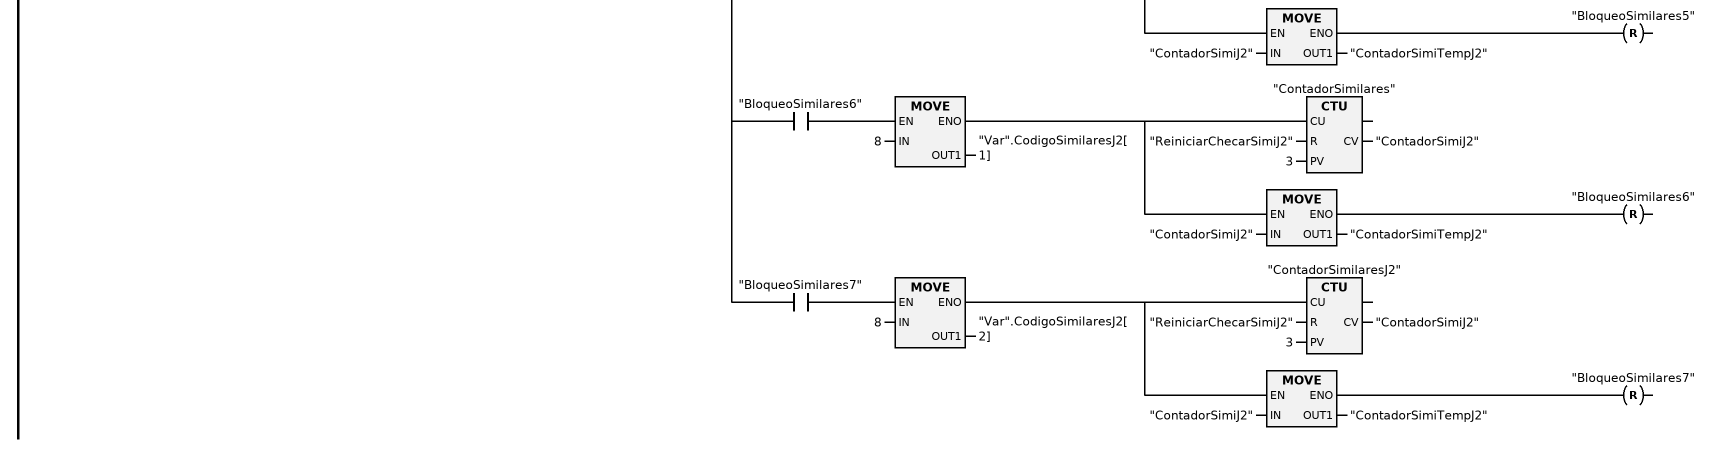
   #_w1 := "Panel1AzulJ2" AND ("Var".VectorPrincipalJ2["IntentoCompletoJ2", 0] = 0) AND "Bounce6";
   IF #_w1 THEN
       "Var".VectorPrincipalJ2["IntentoCompletoJ2", 0] := 5;
       "Intento0J2" := TRUE;
   END_IF;
   #_w2 := #_w1 AND ("Var".VectorPrincipalJ2["IntentoCompletoJ2", 0] = "Var".CodigoOJ2[0]);
   "ContadorCorrectasJ2".CTU(CU := #_w2, R := "ReiniciarChecarCorrJ2", PV := 3, CV => "ContadorCorrJ2");
   IF #_w2 THEN
       "ContadorCorrTempJ2" := "ContadorCorrJ2";
       "Var".CodigoSimilaresJ2[0] := 8;
       "BloqueoSimilares8" := TRUE;
   END_IF;
   #_w3 := #_w2 AND ("Var".CodigoSimilaresJ2[0] = 8);
   "ContadorSimilaresJ2".CTD(CD := #_w3, LD := "ReiniciarChecarSimiJ2", PV := 3, CV => "ContadorSimiJ2");
   IF #_w3 THEN "ContadorSimiTempJ2" := "ContadorSimiJ2"; END_IF;
   #_w4 := #_w1 AND NOT "BloqueoSimilares8" AND ("Var".VectorPrincipalJ2["IntentoCompletoJ2", 0] <> "Var".CodigoOJ2[0]);
   IF #_w4 AND ("Var".VectorPrincipalJ2["IntentoCompletoJ2", 0] = "Var".CodigoSimilaresJ2[1]) THEN
       "BloqueoSimilares5" := TRUE;
   END_IF;
   #_w5 := #_w4 AND ("Var".VectorPrincipalJ2["IntentoCompletoJ2", 0] <> "Var".CodigoSimilaresJ2[1]);
   IF #_w5 AND ("Var".VectorPrincipalJ2["IntentoCompletoJ2", 0] = "Var".CodigoSimilaresJ2[2]) THEN
       "BloqueoSimilares6" := TRUE;
   END_IF;
   IF #_w5 AND ("Var".VectorPrincipalJ2["IntentoCompletoJ2", 0] <> "Var".CodigoSimilaresJ2[2]) AND ("Var".VectorPrincipalJ2["IntentoCompletoJ2", 0] = "Var".CodigoSimilaresJ2[3]) THEN
       "BloqueoSimilares7" := TRUE;
   END_IF;
   #_w6 := #_w1 AND "BloqueoSimilares5";
   IF #_w6 THEN "Var".CodigoSimilaresJ2[1] := 8; END_IF;
   "ContadorSimilaresJ2".CTU(CU := #_w6, R := "ReiniciarChecarSimiJ2", PV := 3, CV => "ContadorSimiJ2");
   IF #_w6 THEN
       "ContadorSimiTempJ2" := "ContadorSimiJ2";
       "BloqueoSimilares5" := FALSE;
   END_IF;
   #_w7 := #_w1 AND "BloqueoSimilares6";
   IF #_w7 THEN "Var".CodigoSimilaresJ2[2] := 8; END_IF;
   "ContadorSimilaresJ2".CTU(CU := #_w7, R := "ReiniciarChecarSimiJ2", PV := 3, CV => "ContadorSimiJ2");
   IF #_w7 THEN
       "ContadorSimiTempJ2" := "ContadorSimiJ2";
       "BloqueoSimilares6" := FALSE;
   END_IF;
   #_w8 := #_w1 AND "BloqueoSimilares7";
   IF #_w8 THEN "Var".CodigoSimilaresJ2[3] := 8; END_IF;
   "ContadorSimilaresJ2".CTU(CU := #_w8, R := "ReiniciarChecarSimiJ2", PV := 3, CV => "ContadorSimiJ2");
   IF #_w8 THEN
       "ContadorSimiTempJ2" := "ContadorSimiJ2";
       "BloqueoSimilares7" := FALSE;
   END_IF;
   #_w9 := "Panel1AzulJ2" AND "Bounce7" AND "Panel1AzulJ2" AND "Intento0J2" AND ("Var".VectorPrincipalJ2["IntentoCompletoJ2", 1] = 0);
   IF #_w9 THEN
       "Var".VectorPrincipalJ2["IntentoCompletoJ2", 1] := 5;
       "Intento1J2" := TRUE;
   END_IF;
   #_w10 := #_w9 AND ("Var".VectorPrincipalJ2["IntentoCompletoJ2", 1] = "Var".CodigoOJ2[1]);
   "ContadorCorrectasJ2".CTU(CU := #_w10, R := "ReiniciarChecarCorrJ2", PV := 3, CV => "ContadorCorrJ2");
   IF #_w10 THEN
       "ContadorCorrTempJ2" := "ContadorCorrJ2";
       "Var".CodigoSimilaresJ2[1] := 8;
       "BloqueoSimilares8" := TRUE;
   END_IF;
   #_w11 := #_w10 AND ("Var".CodigoSimilaresJ2[1] = 8);
   "ContadorSimilaresJ2".CTD(CD := #_w11, LD := "ReiniciarChecarSimiJ2", PV := 3, CV => "ContadorSimiJ2");
   IF #_w11 THEN "ContadorSimiTempJ2" := "ContadorSimiJ2"; END_IF;
   #_w12 := #_w9 AND NOT "BloqueoSimilares8" AND ("Var".VectorPrincipalJ2["IntentoCompletoJ2", 1] <> "Var".CodigoOJ2[1]);
   IF #_w12 AND ("Var".VectorPrincipalJ2["IntentoCompletoJ2", 1] = "Var".CodigoSimilaresJ2[0]) THEN
       "BloqueoSimilares5" := TRUE;
   END_IF;
   #_w13 := #_w12 AND ("Var".VectorPrincipalJ2["IntentoCompletoJ2", 1] <> "Var".CodigoSimilaresJ2[0]);
   IF #_w13 AND ("Var".VectorPrincipalJ2["IntentoCompletoJ2", 1] = "Var".CodigoSimilaresJ2[2]) THEN
       "BloqueoSimilares6" := TRUE;
   END_IF;
   IF #_w13 AND ("Var".VectorPrincipalJ2["IntentoCompletoJ2", 1] <> "Var".CodigoSimilaresJ2[2]) AND ("Var".VectorPrincipalJ2["IntentoCompletoJ2", 1] = "Var".CodigoSimilaresJ2[3]) THEN
       "BloqueoSimilares7" := TRUE;
   END_IF;
   #_w14 := #_w9 AND "BloqueoSimilares5";
   IF #_w14 THEN "Var".CodigoSimilaresJ2[0] := 8; END_IF;
   "ContadorSimilaresJ2".CTU(CU := #_w14, R := "ReiniciarChecarSimiJ2", PV := 3, CV => "ContadorSimiJ2");
   IF #_w14 THEN
       "ContadorSimiTempJ2" := "ContadorSimiJ2";
       "BloqueoSimilares5" := FALSE;
   END_IF;
   #_w15 := #_w9 AND "BloqueoSimilares6";
   IF #_w15 THEN "Var".CodigoSimilaresJ1[2] := 8; END_IF;
   "ContadorSimilaresJ2".CTU(CU := #_w15, R := "ReiniciarChecarSimiJ2", PV := 3, CV => "ContadorSimiJ2");
   IF #_w15 THEN
       "ContadorSimiTempJ2" := "ContadorSimiJ2";
       "BloqueoSimilares6" := FALSE;
   END_IF;
   #_w16 := #_w9 AND "BloqueoSimilares7";
   IF #_w16 THEN "Var".CodigoSimilaresJ2[3] := 8; END_IF;
   "ContadorSimilaresJ2".CTU(CU := #_w16, R := "ReiniciarChecarSimiJ2", PV := 3, CV => "ContadorSimiJ2");
   IF #_w16 THEN
       "ContadorSimiTempJ2" := "ContadorSimiJ2";
       "BloqueoSimilares3" := FALSE;
   END_IF;
   #_w17 := "Panel1AzulJ2" AND "Bounce8" AND "Panel1AzulJ2" AND "Intento1J2" AND ("Var".VectorPrincipalJ2["IntentoCompletoJ2", 2] = 0);
   IF #_w17 THEN
       "Var".VectorPrincipalJ2["IntentoCompletoJ2", 2] := 5;
       "Intento2J2" := TRUE;
   END_IF;
   #_w18 := #_w17 AND ("Var".VectorPrincipalJ2["IntentoCompletoJ2", 2] = "Var".CodigoOJ2[2]);
   "ContadorCorrectasJ2".CTU(CU := #_w18, R := "ReiniciarChecarCorrJ2", PV := 3, CV => "ContadorCorrJ2");
   IF #_w18 THEN
       "ContadorCorrTempJ2" := "ContadorCorrJ2";
       "Var".CodigoSimilaresJ2[2] := 8;
       "BloqueoSimilares8" := TRUE;
   END_IF;
   #_w19 := #_w18 AND ("Var".CodigoSimilaresJ2[2] = 8);
   "ContadorSimilaresJ2".CTD(CD := #_w19, LD := "ReiniciarChecarSimiJ2", PV := 3, CV => "ContadorSimiJ2");
   IF #_w19 THEN "ContadorSimiTempJ2" := "ContadorSimiJ2"; END_IF;
   #_w20 := #_w17 AND NOT "BloqueoSimilares8" AND ("Var".VectorPrincipalJ2["IntentoCompletoJ2", 2] <> "Var".CodigoOJ2[2]);
   IF #_w20 AND ("Var".VectorPrincipalJ2["IntentoCompletoJ2", 2] = "Var".CodigoSimilaresJ2[0]) THEN
       "BloqueoSimilares5" := TRUE;
   END_IF;
   #_w21 := #_w20 AND ("Var".VectorPrincipalJ2["IntentoCompletoJ2", 2] <> "Var".CodigoSimilaresJ2[0]);
   IF #_w21 AND ("Var".VectorPrincipalJ2["IntentoCompletoJ2", 2] = "Var".CodigoSimilaresJ2[1]) THEN
       "BloqueoSimilares6" := TRUE;
   END_IF;
   IF #_w21 AND ("Var".VectorPrincipalJ2["IntentoCompletoJ2", 2] <> "Var".CodigoSimilaresJ2[1]) AND ("Var".VectorPrincipalJ2["IntentoCompletoJ2", 2] = "Var".CodigoSimilaresJ2[3]) THEN
       "BloqueoSimilares7" := TRUE;
   END_IF;
   #_w22 := #_w17 AND "BloqueoSimilares5";
   IF #_w22 THEN "Var".CodigoSimilaresJ2[0] := 8; END_IF;
   "ContadorSimilaresJ2".CTU(CU := #_w22, R := "ReiniciarChecarSimiJ2", PV := 3, CV => "ContadorSimiJ2");
   IF #_w22 THEN
       "ContadorSimiTempJ2" := "ContadorSimiJ2";
       "BloqueoSimilares5" := FALSE;
   END_IF;
   #_w23 := #_w17 AND "BloqueoSimilares6";
   IF #_w23 THEN "Var".CodigoSimilaresJ2[1] := 8; END_IF;
   "ContadorSimilaresJ2".CTU(CU := #_w23, R := "ReiniciarChecarSimiJ2", PV := 3, CV => "ContadorSimiJ2");
   IF #_w23 THEN
       "ContadorSimiTempJ2" := "ContadorSimiJ2";
       "BloqueoSimilares6" := FALSE;
   END_IF;
   #_w24 := #_w17 AND "BloqueoSimilares7";
   IF #_w24 THEN "Var".CodigoSimilaresJ2[3] := 8; END_IF;
   "ContadorSimilaresJ2".CTU(CU := #_w24, R := "ReiniciarChecarSimiJ2", PV := 3, CV => "ContadorSimiJ2");
   IF #_w24 THEN
       "ContadorSimiTempJ2" := "ContadorSimiJ2";
       "BloqueoSimilares7" := FALSE;
   END_IF;
   #_w25 := "Panel1AzulJ2" AND "Bounce9" AND "Panel1AzulJ2" AND "Intento2J2" AND ("Var".VectorPrincipalJ2["IntentoCompletoJ2", 3] = 0);
   IF #_w25 THEN
       "Var".VectorPrincipalJ2["IntentoCompletoJ2", 3] := 5;
       "Intento3J2" := TRUE;
   END_IF;
   #_w26 := #_w25 AND ("Var".VectorPrincipalJ2["IntentoCompletoJ2", 3] = "Var".CodigoOJ2[3]);
   "ContadorCorrectasJ2".CTU(CU := #_w26, R := "ReiniciarChecarCorrJ2", PV := 3, CV => "ContadorCorrJ2");
   IF #_w26 THEN
       "ContadorCorrTempJ2" := "ContadorCorrJ2";
       "Var".CodigoSimilaresJ2[3] := 8;
       "BloqueoSimilares8" := TRUE;
   END_IF;
   #_w27 := #_w26 AND ("Var".CodigoSimilaresJ2[3] = 8);
   "ContadorSimilaresJ2".CTD(CD := #_w27, LD := "ReiniciarChecarSimiJ2", PV := 3, CV => "ContadorSimiJ2");
   IF #_w27 THEN "ContadorSimiTempJ2" := "ContadorSimiJ2"; END_IF;
   #_w28 := #_w25 AND NOT "BloqueoSimilares8" AND ("Var".VectorPrincipalJ2["IntentoCompletoJ2", 3] <> "Var".CodigoOJ2[3]);
   IF #_w28 AND ("Var".VectorPrincipalJ2["IntentoCompletoJ2", 3] = "Var".CodigoSimilaresJ2[0]) THEN
       "BloqueoSimilares5" := TRUE;
   END_IF;
   #_w29 := #_w28 AND ("Var".VectorPrincipalJ2["IntentoCompletoJ2", 3] <> "Var".CodigoSimilaresJ2[0]);
   IF #_w29 AND ("Var".VectorPrincipalJ2["IntentoCompletoJ2", 3] = "Var".CodigoSimilaresJ2[1]) THEN
       "BloqueoSimilares6" := TRUE;
   END_IF;
   IF #_w29 AND ("Var".VectorPrincipalJ2["IntentoCompletoJ2", 3] <> "Var".CodigoSimilaresJ2[1]) AND ("Var".VectorPrincipalJ2["IntentoCompletoJ2", 3] = "Var".CodigoSimilaresJ2[2]) THEN
       "BloqueoSimilares7" := TRUE;
   END_IF;
   #_w30 := #_w25 AND "BloqueoSimilares5";
   IF #_w30 THEN "Var".CodigoSimilaresJ2[0] := 8; END_IF;
   "ContadorSimilaresJ2".CTU(CU := #_w30, R := "ReiniciarChecarSimiJ2", PV := 3, CV => "ContadorSimiJ2");
   IF #_w30 THEN
       "ContadorSimiTempJ2" := "ContadorSimiJ2";
       "BloqueoSimilares5" := FALSE;
   END_IF;
   #_w31 := #_w25 AND "BloqueoSimilares6";
   IF #_w31 THEN "Var".CodigoSimilaresJ2[1] := 8; END_IF;
   "ContadorSimilares".CTU(CU := #_w31, R := "ReiniciarChecarSimiJ2", PV := 3, CV => "ContadorSimiJ2");
   IF #_w31 THEN
       "ContadorSimiTempJ2" := "ContadorSimiJ2";
       "BloqueoSimilares6" := FALSE;
   END_IF;
   #_w32 := #_w25 AND "BloqueoSimilares7";
   IF #_w32 THEN "Var".CodigoSimilaresJ2[2] := 8; END_IF;
   "ContadorSimilaresJ2".CTU(CU := #_w32, R := "ReiniciarChecarSimiJ2", PV := 3, CV => "ContadorSimiJ2");
   IF #_w32 THEN
       "ContadorSimiTempJ2" := "ContadorSimiJ2";
       "BloqueoSimilares7" := FALSE;
   END_IF;
END_REGION

REGION Network 24: Verde J2
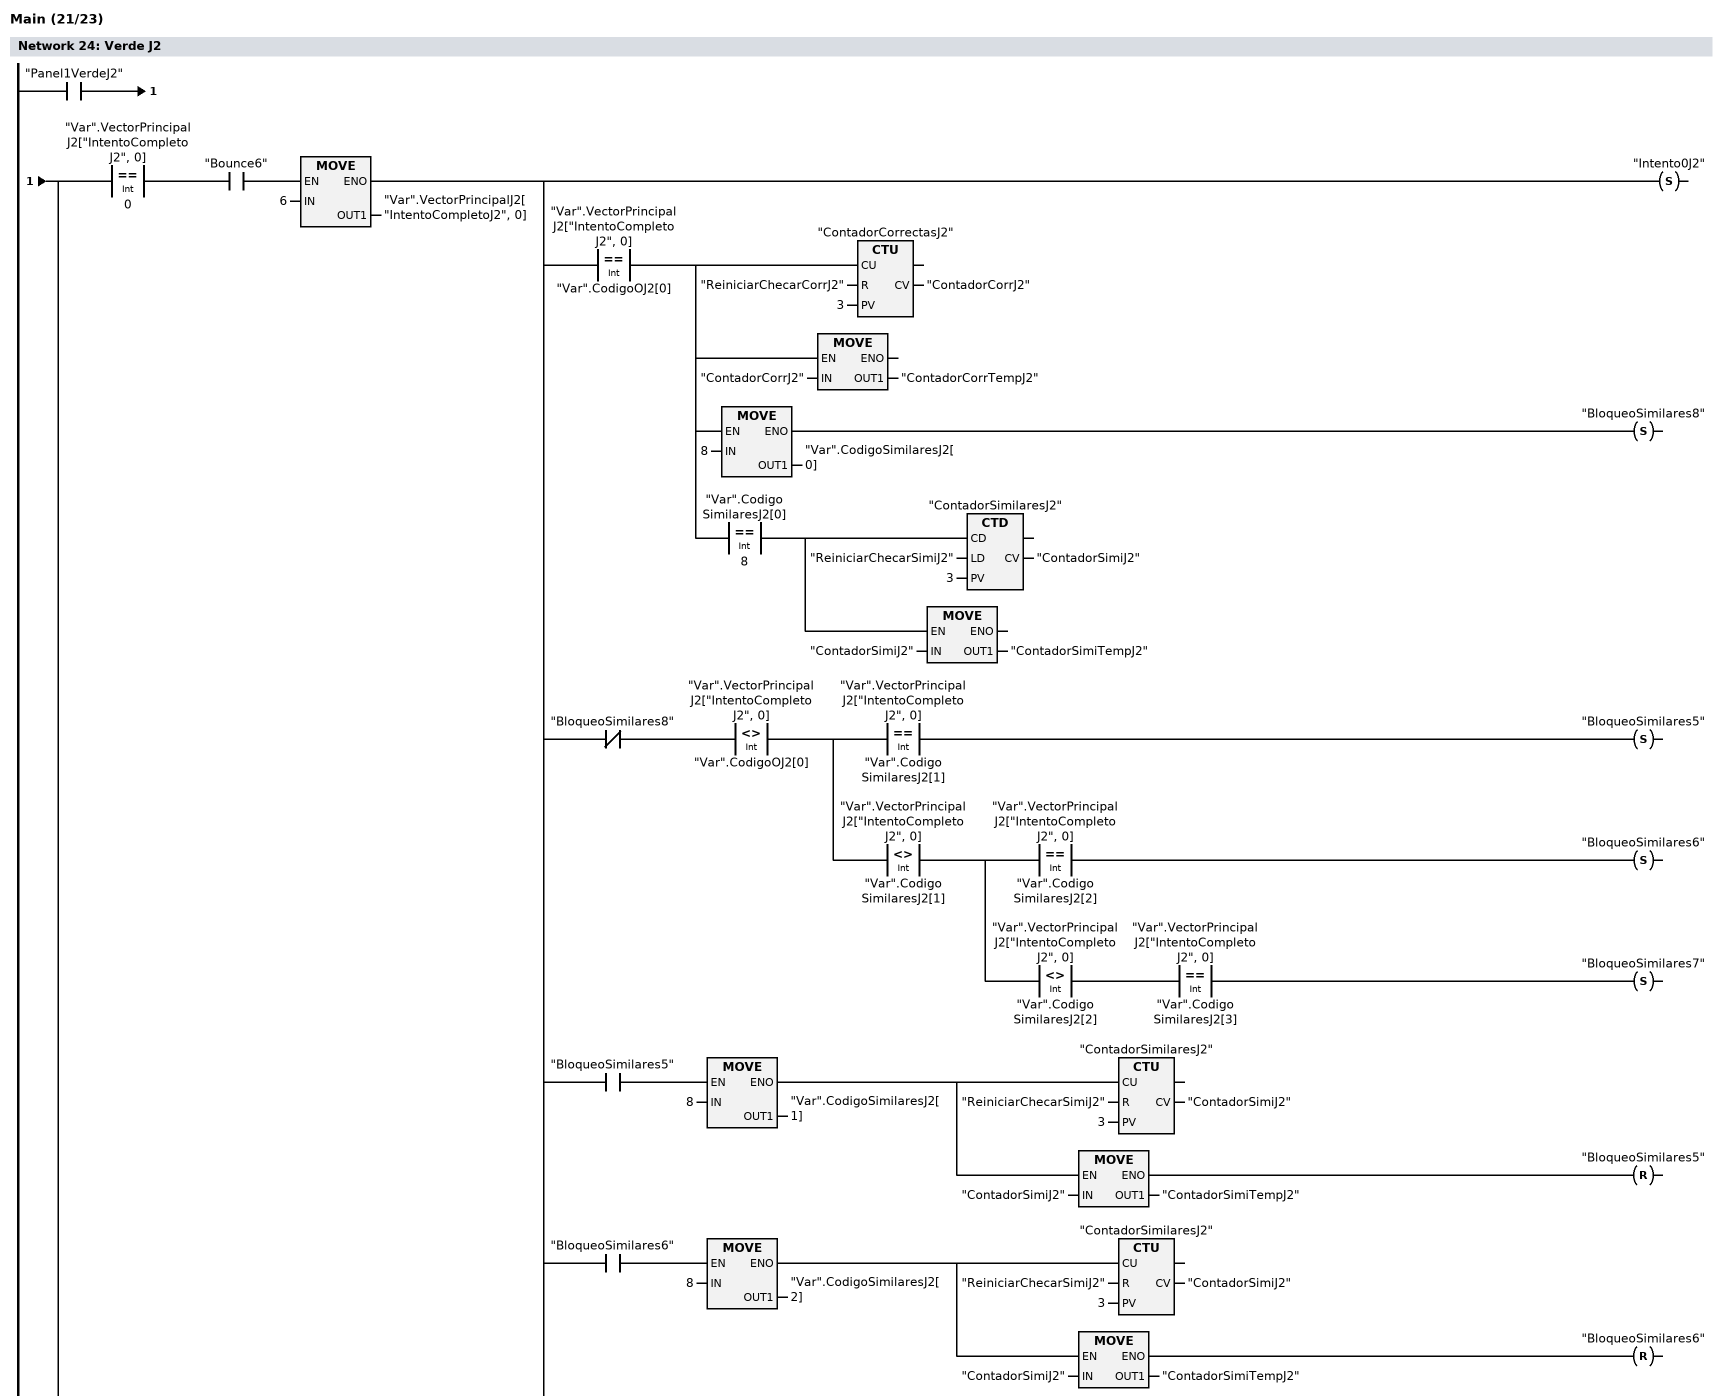
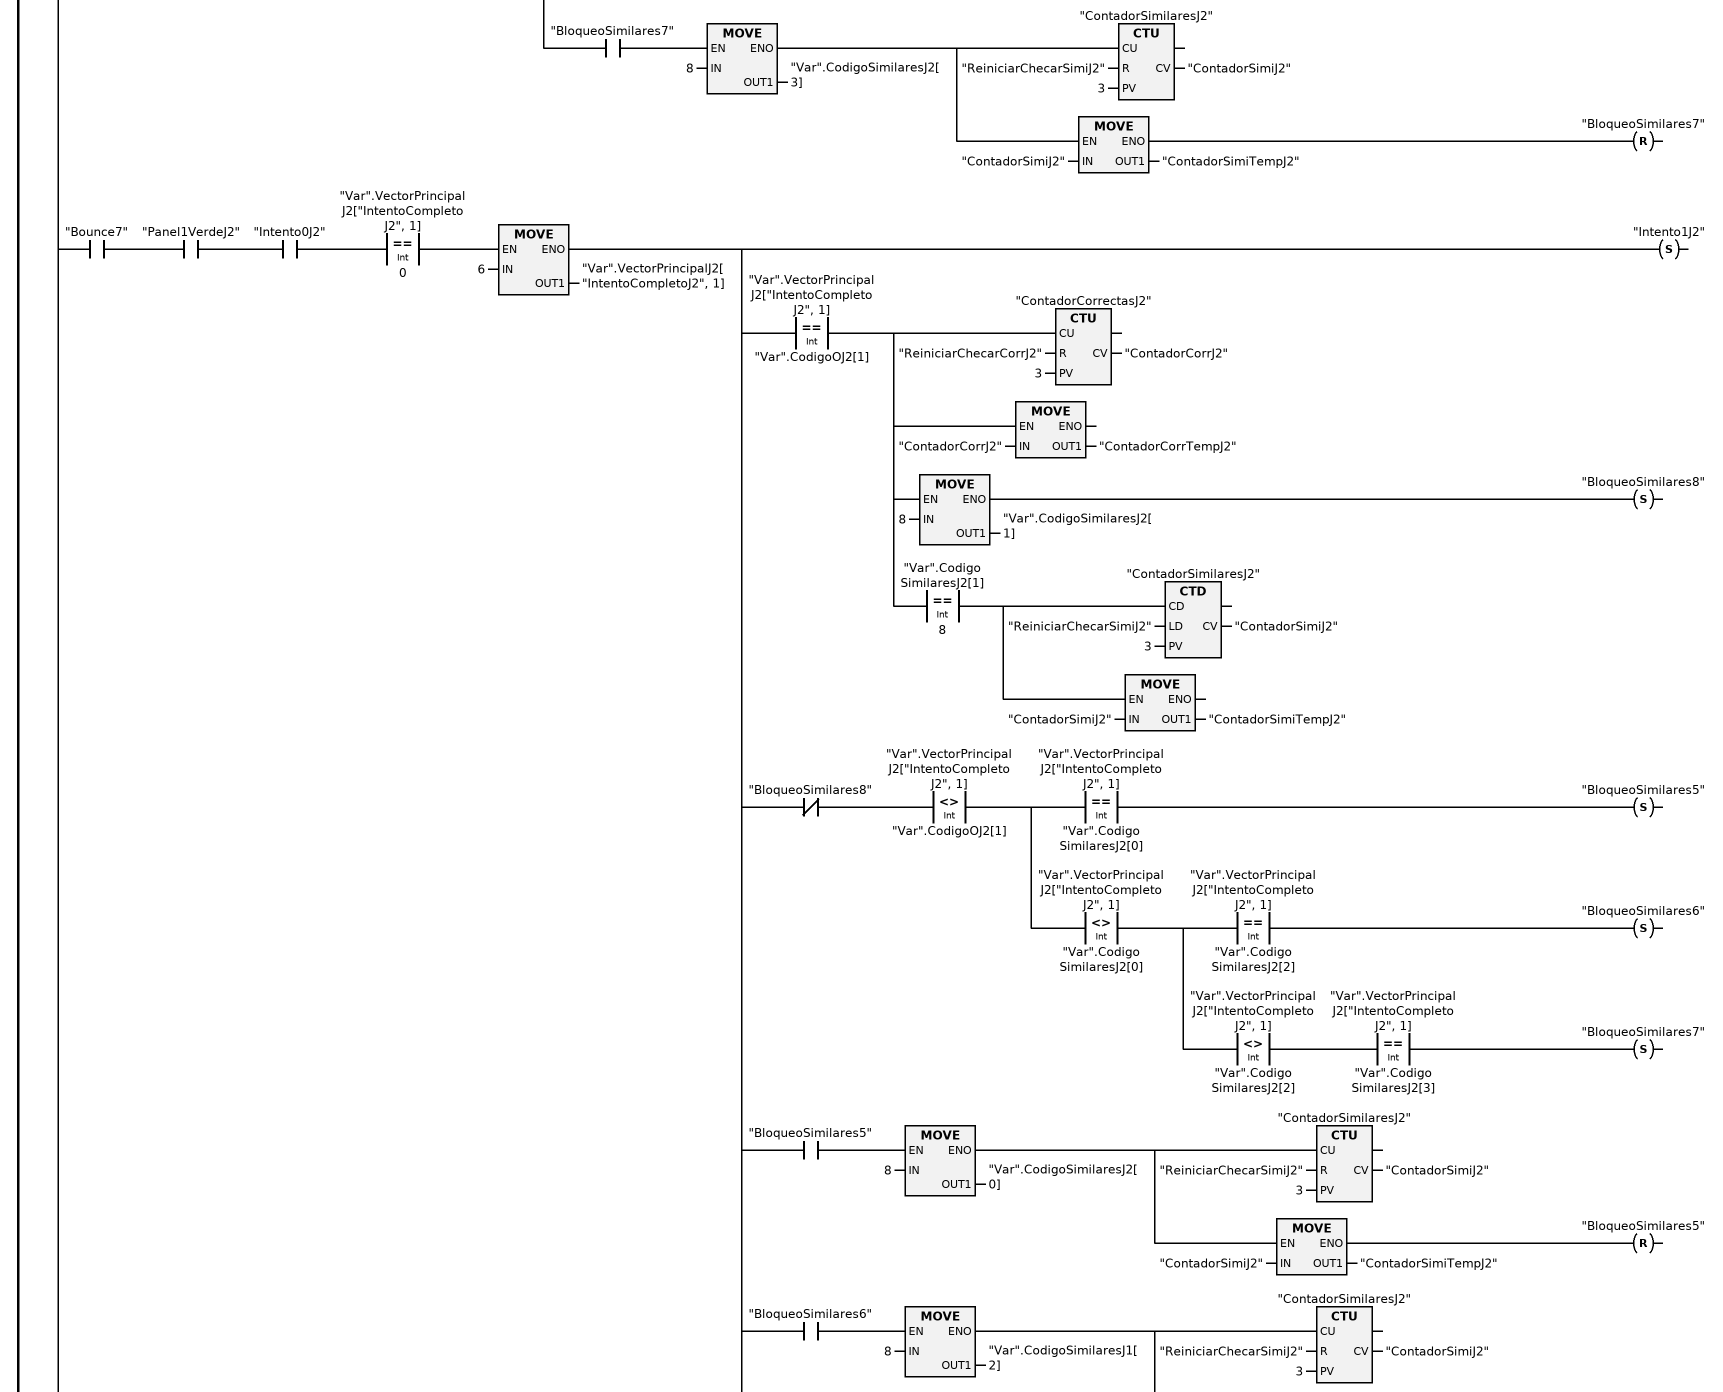
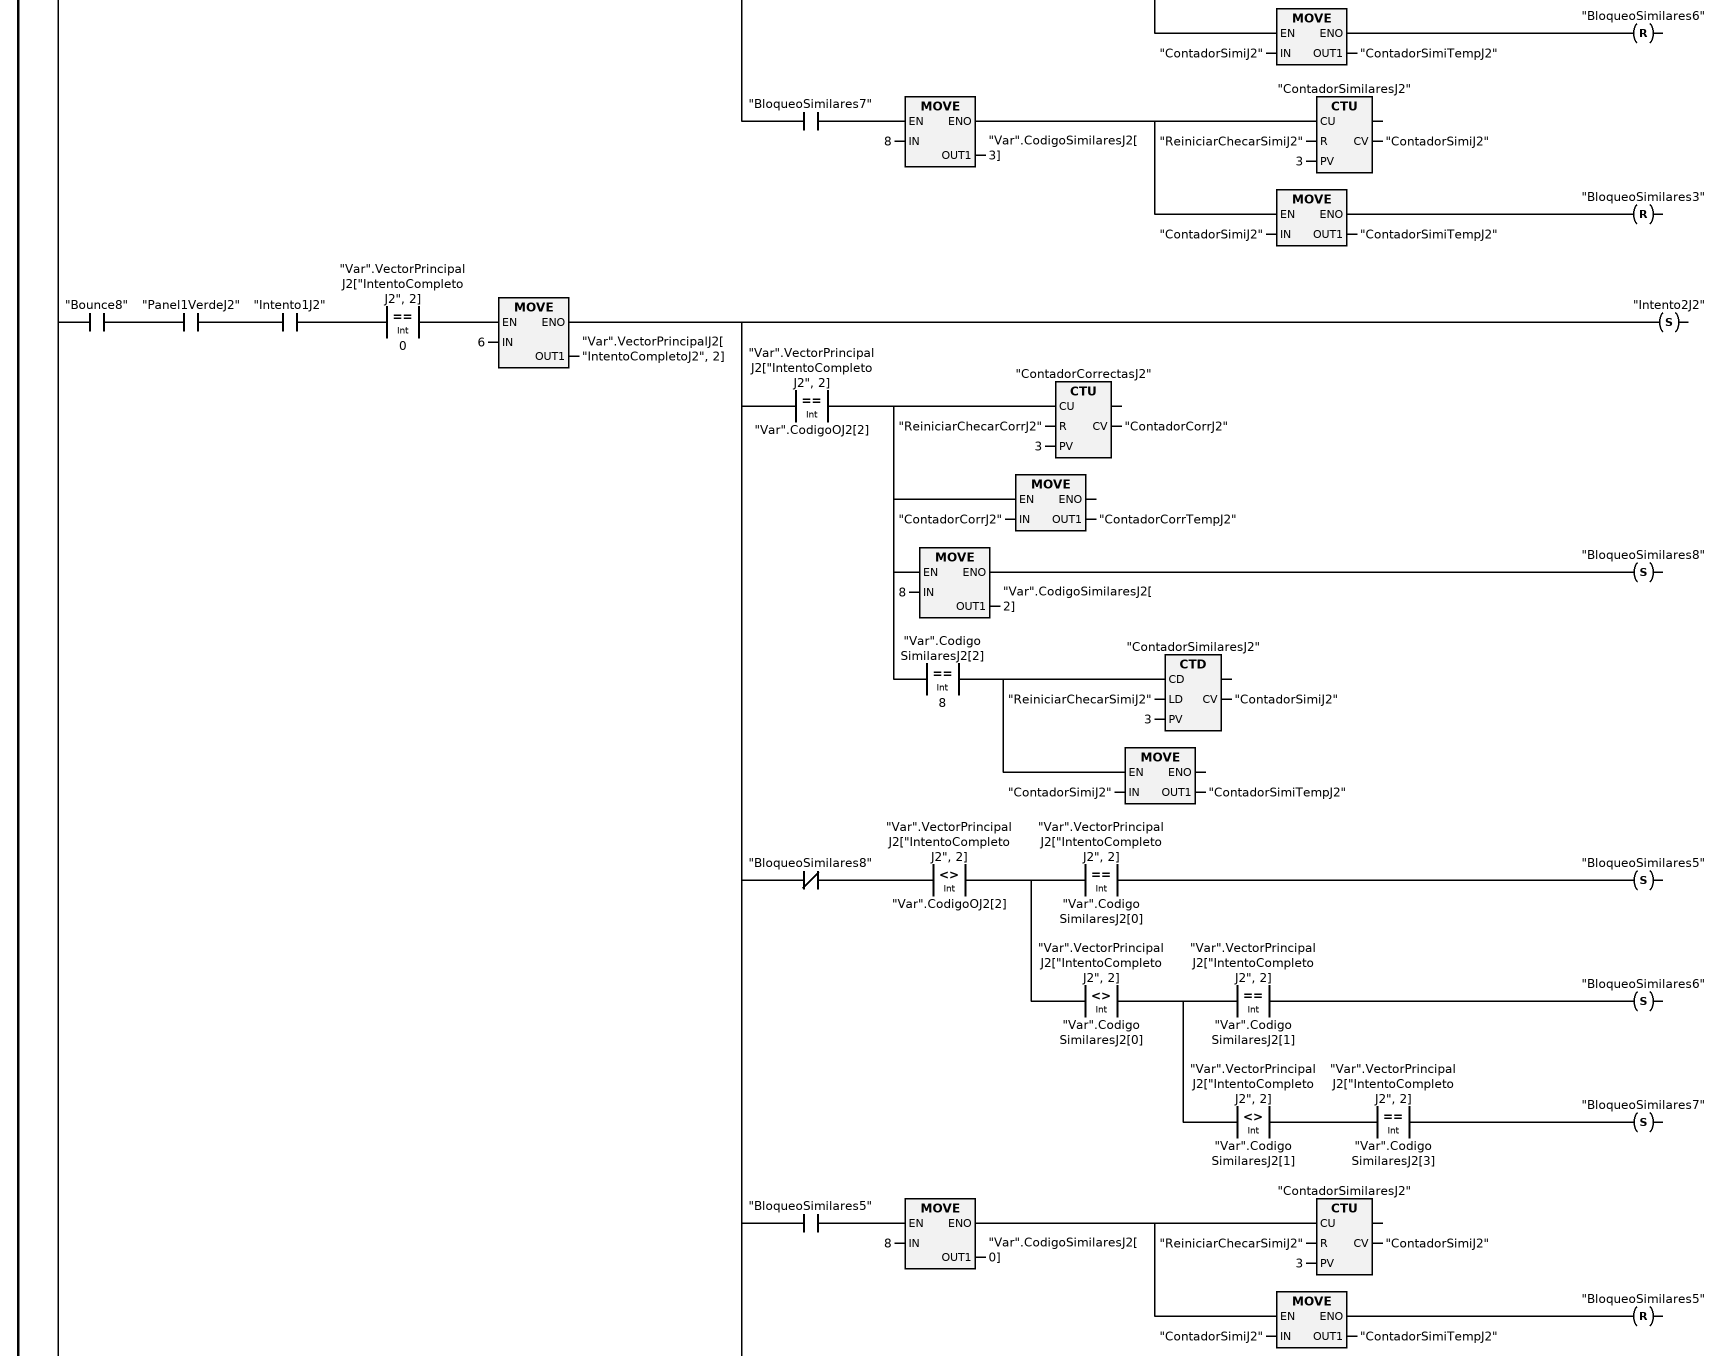
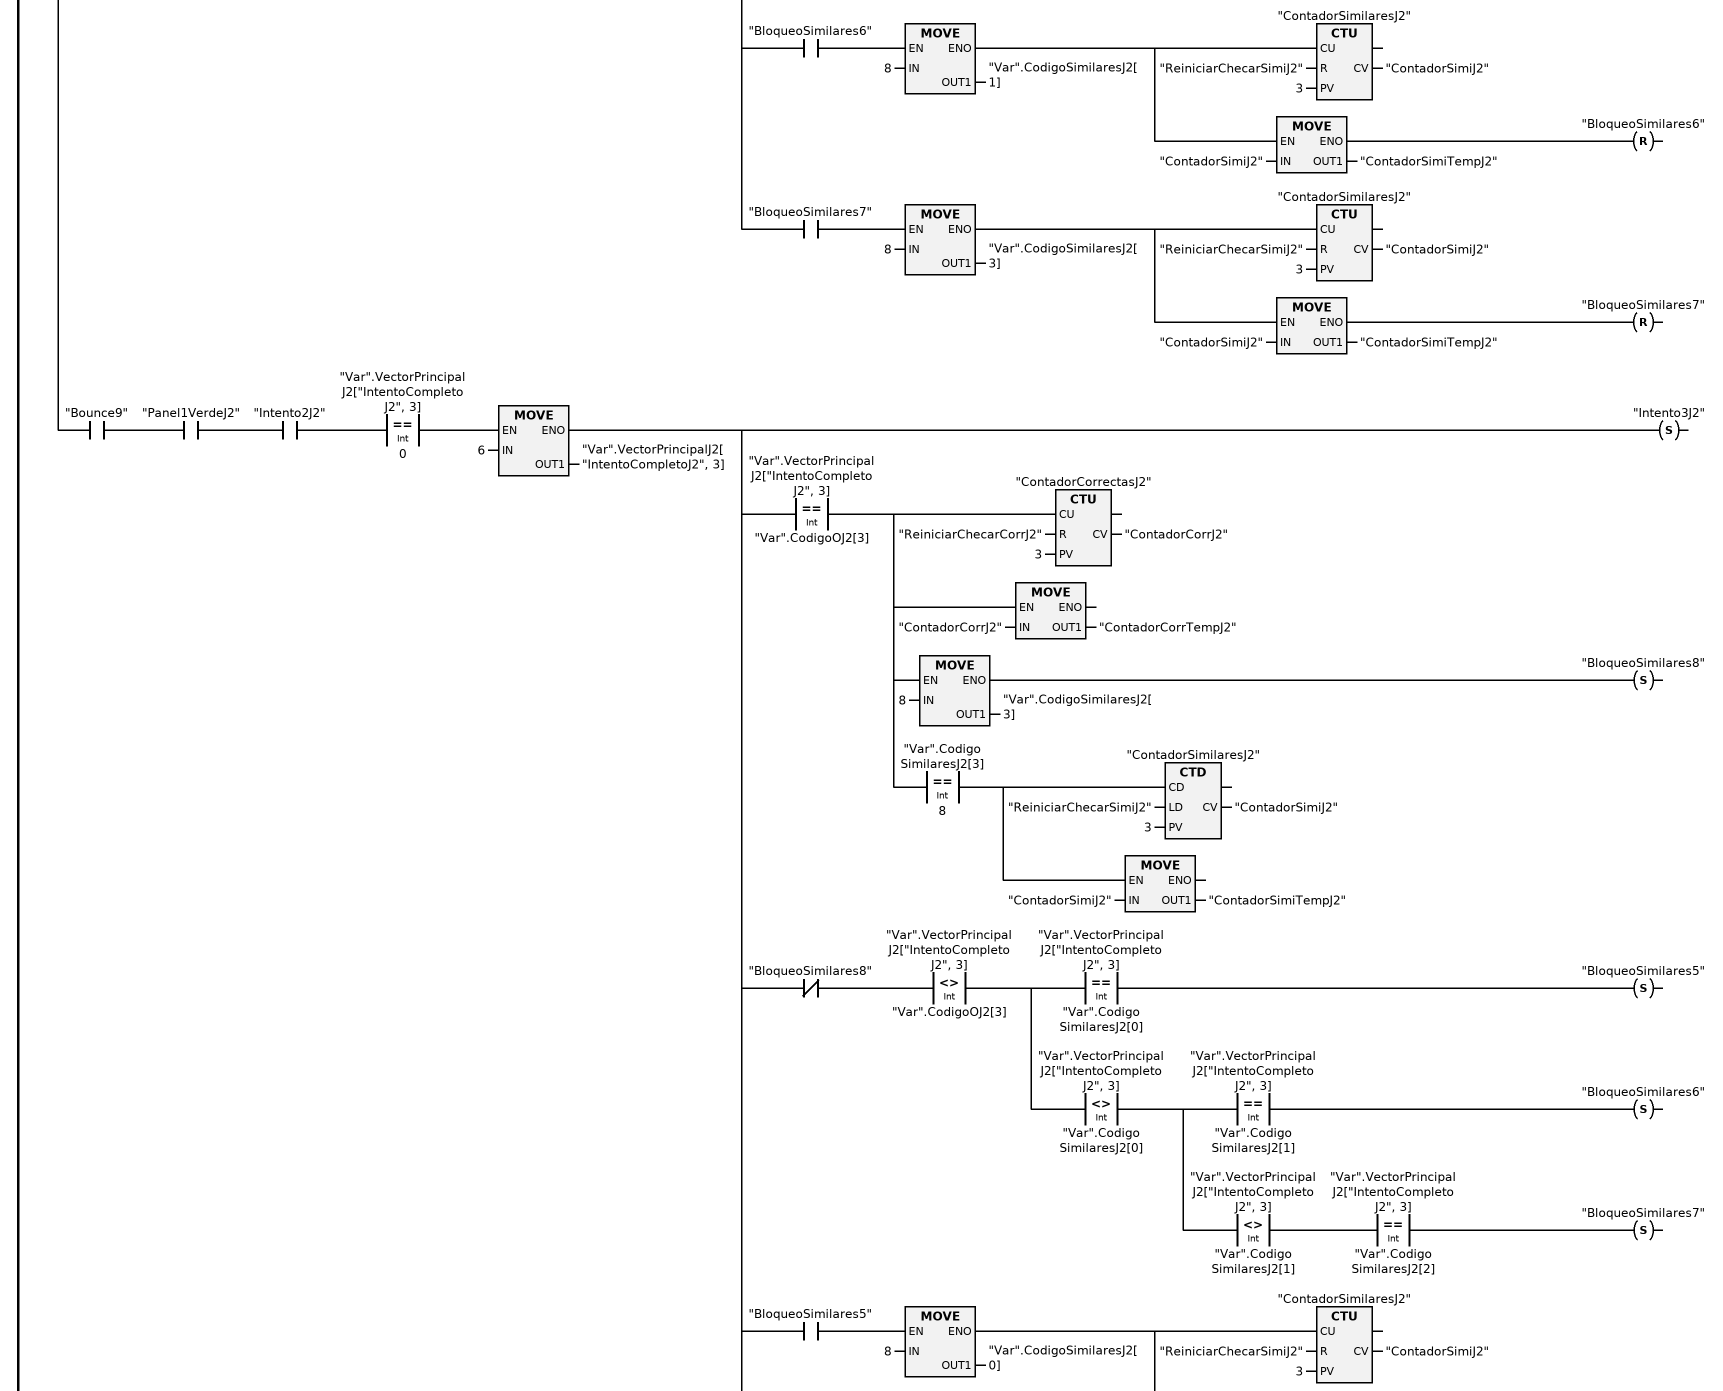
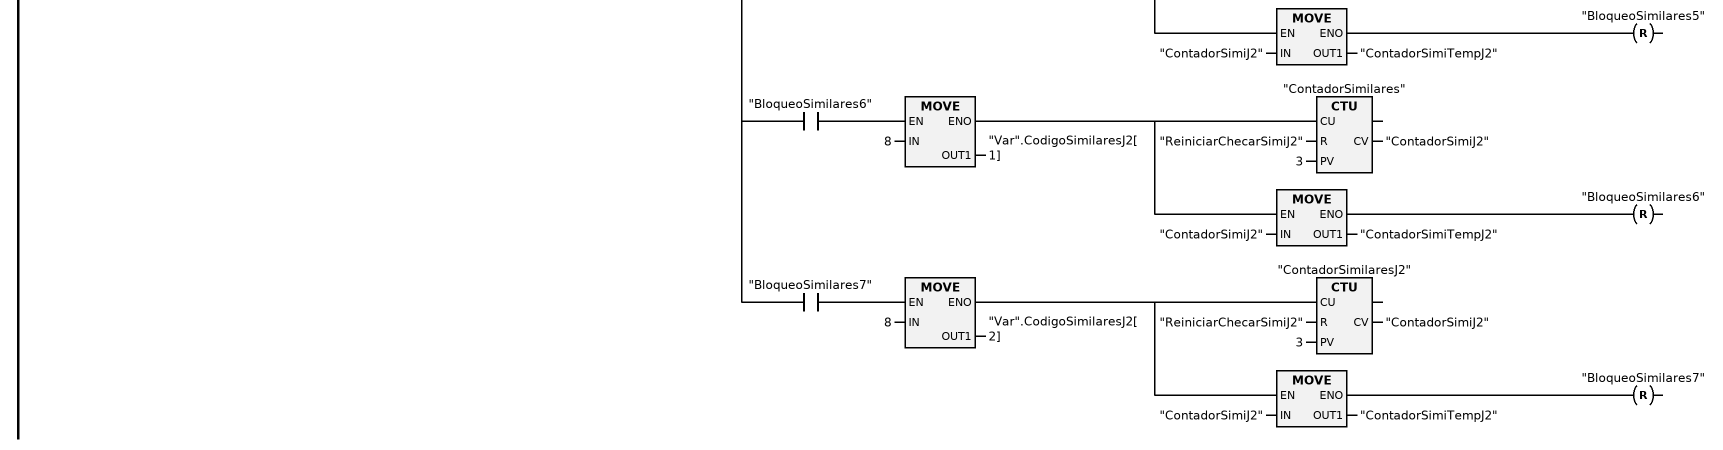
   #_w1 := "Panel1VerdeJ2" AND ("Var".VectorPrincipalJ2["IntentoCompletoJ2", 0] = 0) AND "Bounce6";
   IF #_w1 THEN
       "Var".VectorPrincipalJ2["IntentoCompletoJ2", 0] := 6;
       "Intento0J2" := TRUE;
   END_IF;
   #_w2 := #_w1 AND ("Var".VectorPrincipalJ2["IntentoCompletoJ2", 0] = "Var".CodigoOJ2[0]);
   "ContadorCorrectasJ2".CTU(CU := #_w2, R := "ReiniciarChecarCorrJ2", PV := 3, CV => "ContadorCorrJ2");
   IF #_w2 THEN
       "ContadorCorrTempJ2" := "ContadorCorrJ2";
       "Var".CodigoSimilaresJ2[0] := 8;
       "BloqueoSimilares8" := TRUE;
   END_IF;
   #_w3 := #_w2 AND ("Var".CodigoSimilaresJ2[0] = 8);
   "ContadorSimilaresJ2".CTD(CD := #_w3, LD := "ReiniciarChecarSimiJ2", PV := 3, CV => "ContadorSimiJ2");
   IF #_w3 THEN "ContadorSimiTempJ2" := "ContadorSimiJ2"; END_IF;
   #_w4 := #_w1 AND NOT "BloqueoSimilares8" AND ("Var".VectorPrincipalJ2["IntentoCompletoJ2", 0] <> "Var".CodigoOJ2[0]);
   IF #_w4 AND ("Var".VectorPrincipalJ2["IntentoCompletoJ2", 0] = "Var".CodigoSimilaresJ2[1]) THEN
       "BloqueoSimilares5" := TRUE;
   END_IF;
   #_w5 := #_w4 AND ("Var".VectorPrincipalJ2["IntentoCompletoJ2", 0] <> "Var".CodigoSimilaresJ2[1]);
   IF #_w5 AND ("Var".VectorPrincipalJ2["IntentoCompletoJ2", 0] = "Var".CodigoSimilaresJ2[2]) THEN
       "BloqueoSimilares6" := TRUE;
   END_IF;
   IF #_w5 AND ("Var".VectorPrincipalJ2["IntentoCompletoJ2", 0] <> "Var".CodigoSimilaresJ2[2]) AND ("Var".VectorPrincipalJ2["IntentoCompletoJ2", 0] = "Var".CodigoSimilaresJ2[3]) THEN
       "BloqueoSimilares7" := TRUE;
   END_IF;
   #_w6 := #_w1 AND "BloqueoSimilares5";
   IF #_w6 THEN "Var".CodigoSimilaresJ2[1] := 8; END_IF;
   "ContadorSimilaresJ2".CTU(CU := #_w6, R := "ReiniciarChecarSimiJ2", PV := 3, CV => "ContadorSimiJ2");
   IF #_w6 THEN
       "ContadorSimiTempJ2" := "ContadorSimiJ2";
       "BloqueoSimilares5" := FALSE;
   END_IF;
   #_w7 := #_w1 AND "BloqueoSimilares6";
   IF #_w7 THEN "Var".CodigoSimilaresJ2[2] := 8; END_IF;
   "ContadorSimilaresJ2".CTU(CU := #_w7, R := "ReiniciarChecarSimiJ2", PV := 3, CV => "ContadorSimiJ2");
   IF #_w7 THEN
       "ContadorSimiTempJ2" := "ContadorSimiJ2";
       "BloqueoSimilares6" := FALSE;
   END_IF;
   #_w8 := #_w1 AND "BloqueoSimilares7";
   IF #_w8 THEN "Var".CodigoSimilaresJ2[3] := 8; END_IF;
   "ContadorSimilaresJ2".CTU(CU := #_w8, R := "ReiniciarChecarSimiJ2", PV := 3, CV => "ContadorSimiJ2");
   IF #_w8 THEN
       "ContadorSimiTempJ2" := "ContadorSimiJ2";
       "BloqueoSimilares7" := FALSE;
   END_IF;
   #_w9 := "Panel1VerdeJ2" AND "Bounce7" AND "Panel1VerdeJ2" AND "Intento0J2" AND ("Var".VectorPrincipalJ2["IntentoCompletoJ2", 1] = 0);
   IF #_w9 THEN
       "Var".VectorPrincipalJ2["IntentoCompletoJ2", 1] := 6;
       "Intento1J2" := TRUE;
   END_IF;
   #_w10 := #_w9 AND ("Var".VectorPrincipalJ2["IntentoCompletoJ2", 1] = "Var".CodigoOJ2[1]);
   "ContadorCorrectasJ2".CTU(CU := #_w10, R := "ReiniciarChecarCorrJ2", PV := 3, CV => "ContadorCorrJ2");
   IF #_w10 THEN
       "ContadorCorrTempJ2" := "ContadorCorrJ2";
       "Var".CodigoSimilaresJ2[1] := 8;
       "BloqueoSimilares8" := TRUE;
   END_IF;
   #_w11 := #_w10 AND ("Var".CodigoSimilaresJ2[1] = 8);
   "ContadorSimilaresJ2".CTD(CD := #_w11, LD := "ReiniciarChecarSimiJ2", PV := 3, CV => "ContadorSimiJ2");
   IF #_w11 THEN "ContadorSimiTempJ2" := "ContadorSimiJ2"; END_IF;
   #_w12 := #_w9 AND NOT "BloqueoSimilares8" AND ("Var".VectorPrincipalJ2["IntentoCompletoJ2", 1] <> "Var".CodigoOJ2[1]);
   IF #_w12 AND ("Var".VectorPrincipalJ2["IntentoCompletoJ2", 1] = "Var".CodigoSimilaresJ2[0]) THEN
       "BloqueoSimilares5" := TRUE;
   END_IF;
   #_w13 := #_w12 AND ("Var".VectorPrincipalJ2["IntentoCompletoJ2", 1] <> "Var".CodigoSimilaresJ2[0]);
   IF #_w13 AND ("Var".VectorPrincipalJ2["IntentoCompletoJ2", 1] = "Var".CodigoSimilaresJ2[2]) THEN
       "BloqueoSimilares6" := TRUE;
   END_IF;
   IF #_w13 AND ("Var".VectorPrincipalJ2["IntentoCompletoJ2", 1] <> "Var".CodigoSimilaresJ2[2]) AND ("Var".VectorPrincipalJ2["IntentoCompletoJ2", 1] = "Var".CodigoSimilaresJ2[3]) THEN
       "BloqueoSimilares7" := TRUE;
   END_IF;
   #_w14 := #_w9 AND "BloqueoSimilares5";
   IF #_w14 THEN "Var".CodigoSimilaresJ2[0] := 8; END_IF;
   "ContadorSimilaresJ2".CTU(CU := #_w14, R := "ReiniciarChecarSimiJ2", PV := 3, CV => "ContadorSimiJ2");
   IF #_w14 THEN
       "ContadorSimiTempJ2" := "ContadorSimiJ2";
       "BloqueoSimilares5" := FALSE;
   END_IF;
   #_w15 := #_w9 AND "BloqueoSimilares6";
   IF #_w15 THEN "Var".CodigoSimilaresJ1[2] := 8; END_IF;
   "ContadorSimilaresJ2".CTU(CU := #_w15, R := "ReiniciarChecarSimiJ2", PV := 3, CV => "ContadorSimiJ2");
   IF #_w15 THEN
       "ContadorSimiTempJ2" := "ContadorSimiJ2";
       "BloqueoSimilares6" := FALSE;
   END_IF;
   #_w16 := #_w9 AND "BloqueoSimilares7";
   IF #_w16 THEN "Var".CodigoSimilaresJ2[3] := 8; END_IF;
   "ContadorSimilaresJ2".CTU(CU := #_w16, R := "ReiniciarChecarSimiJ2", PV := 3, CV => "ContadorSimiJ2");
   IF #_w16 THEN
       "ContadorSimiTempJ2" := "ContadorSimiJ2";
       "BloqueoSimilares3" := FALSE;
   END_IF;
   #_w17 := "Panel1VerdeJ2" AND "Bounce8" AND "Panel1VerdeJ2" AND "Intento1J2" AND ("Var".VectorPrincipalJ2["IntentoCompletoJ2", 2] = 0);
   IF #_w17 THEN
       "Var".VectorPrincipalJ2["IntentoCompletoJ2", 2] := 6;
       "Intento2J2" := TRUE;
   END_IF;
   #_w18 := #_w17 AND ("Var".VectorPrincipalJ2["IntentoCompletoJ2", 2] = "Var".CodigoOJ2[2]);
   "ContadorCorrectasJ2".CTU(CU := #_w18, R := "ReiniciarChecarCorrJ2", PV := 3, CV => "ContadorCorrJ2");
   IF #_w18 THEN
       "ContadorCorrTempJ2" := "ContadorCorrJ2";
       "Var".CodigoSimilaresJ2[2] := 8;
       "BloqueoSimilares8" := TRUE;
   END_IF;
   #_w19 := #_w18 AND ("Var".CodigoSimilaresJ2[2] = 8);
   "ContadorSimilaresJ2".CTD(CD := #_w19, LD := "ReiniciarChecarSimiJ2", PV := 3, CV => "ContadorSimiJ2");
   IF #_w19 THEN "ContadorSimiTempJ2" := "ContadorSimiJ2"; END_IF;
   #_w20 := #_w17 AND NOT "BloqueoSimilares8" AND ("Var".VectorPrincipalJ2["IntentoCompletoJ2", 2] <> "Var".CodigoOJ2[2]);
   IF #_w20 AND ("Var".VectorPrincipalJ2["IntentoCompletoJ2", 2] = "Var".CodigoSimilaresJ2[0]) THEN
       "BloqueoSimilares5" := TRUE;
   END_IF;
   #_w21 := #_w20 AND ("Var".VectorPrincipalJ2["IntentoCompletoJ2", 2] <> "Var".CodigoSimilaresJ2[0]);
   IF #_w21 AND ("Var".VectorPrincipalJ2["IntentoCompletoJ2", 2] = "Var".CodigoSimilaresJ2[1]) THEN
       "BloqueoSimilares6" := TRUE;
   END_IF;
   IF #_w21 AND ("Var".VectorPrincipalJ2["IntentoCompletoJ2", 2] <> "Var".CodigoSimilaresJ2[1]) AND ("Var".VectorPrincipalJ2["IntentoCompletoJ2", 2] = "Var".CodigoSimilaresJ2[3]) THEN
       "BloqueoSimilares7" := TRUE;
   END_IF;
   #_w22 := #_w17 AND "BloqueoSimilares5";
   IF #_w22 THEN "Var".CodigoSimilaresJ2[0] := 8; END_IF;
   "ContadorSimilaresJ2".CTU(CU := #_w22, R := "ReiniciarChecarSimiJ2", PV := 3, CV => "ContadorSimiJ2");
   IF #_w22 THEN
       "ContadorSimiTempJ2" := "ContadorSimiJ2";
       "BloqueoSimilares5" := FALSE;
   END_IF;
   #_w23 := #_w17 AND "BloqueoSimilares6";
   IF #_w23 THEN "Var".CodigoSimilaresJ2[1] := 8; END_IF;
   "ContadorSimilaresJ2".CTU(CU := #_w23, R := "ReiniciarChecarSimiJ2", PV := 3, CV => "ContadorSimiJ2");
   IF #_w23 THEN
       "ContadorSimiTempJ2" := "ContadorSimiJ2";
       "BloqueoSimilares6" := FALSE;
   END_IF;
   #_w24 := #_w17 AND "BloqueoSimilares7";
   IF #_w24 THEN "Var".CodigoSimilaresJ2[3] := 8; END_IF;
   "ContadorSimilaresJ2".CTU(CU := #_w24, R := "ReiniciarChecarSimiJ2", PV := 3, CV => "ContadorSimiJ2");
   IF #_w24 THEN
       "ContadorSimiTempJ2" := "ContadorSimiJ2";
       "BloqueoSimilares7" := FALSE;
   END_IF;
   #_w25 := "Panel1VerdeJ2" AND "Bounce9" AND "Panel1VerdeJ2" AND "Intento2J2" AND ("Var".VectorPrincipalJ2["IntentoCompletoJ2", 3] = 0);
   IF #_w25 THEN
       "Var".VectorPrincipalJ2["IntentoCompletoJ2", 3] := 6;
       "Intento3J2" := TRUE;
   END_IF;
   #_w26 := #_w25 AND ("Var".VectorPrincipalJ2["IntentoCompletoJ2", 3] = "Var".CodigoOJ2[3]);
   "ContadorCorrectasJ2".CTU(CU := #_w26, R := "ReiniciarChecarCorrJ2", PV := 3, CV => "ContadorCorrJ2");
   IF #_w26 THEN
       "ContadorCorrTempJ2" := "ContadorCorrJ2";
       "Var".CodigoSimilaresJ2[3] := 8;
       "BloqueoSimilares8" := TRUE;
   END_IF;
   #_w27 := #_w26 AND ("Var".CodigoSimilaresJ2[3] = 8);
   "ContadorSimilaresJ2".CTD(CD := #_w27, LD := "ReiniciarChecarSimiJ2", PV := 3, CV => "ContadorSimiJ2");
   IF #_w27 THEN "ContadorSimiTempJ2" := "ContadorSimiJ2"; END_IF;
   #_w28 := #_w25 AND NOT "BloqueoSimilares8" AND ("Var".VectorPrincipalJ2["IntentoCompletoJ2", 3] <> "Var".CodigoOJ2[3]);
   IF #_w28 AND ("Var".VectorPrincipalJ2["IntentoCompletoJ2", 3] = "Var".CodigoSimilaresJ2[0]) THEN
       "BloqueoSimilares5" := TRUE;
   END_IF;
   #_w29 := #_w28 AND ("Var".VectorPrincipalJ2["IntentoCompletoJ2", 3] <> "Var".CodigoSimilaresJ2[0]);
   IF #_w29 AND ("Var".VectorPrincipalJ2["IntentoCompletoJ2", 3] = "Var".CodigoSimilaresJ2[1]) THEN
       "BloqueoSimilares6" := TRUE;
   END_IF;
   IF #_w29 AND ("Var".VectorPrincipalJ2["IntentoCompletoJ2", 3] <> "Var".CodigoSimilaresJ2[1]) AND ("Var".VectorPrincipalJ2["IntentoCompletoJ2", 3] = "Var".CodigoSimilaresJ2[2]) THEN
       "BloqueoSimilares7" := TRUE;
   END_IF;
   #_w30 := #_w25 AND "BloqueoSimilares5";
   IF #_w30 THEN "Var".CodigoSimilaresJ2[0] := 8; END_IF;
   "ContadorSimilaresJ2".CTU(CU := #_w30, R := "ReiniciarChecarSimiJ2", PV := 3, CV => "ContadorSimiJ2");
   IF #_w30 THEN
       "ContadorSimiTempJ2" := "ContadorSimiJ2";
       "BloqueoSimilares5" := FALSE;
   END_IF;
   #_w31 := #_w25 AND "BloqueoSimilares6";
   IF #_w31 THEN "Var".CodigoSimilaresJ2[1] := 8; END_IF;
   "ContadorSimilares".CTU(CU := #_w31, R := "ReiniciarChecarSimiJ2", PV := 3, CV => "ContadorSimiJ2");
   IF #_w31 THEN
       "ContadorSimiTempJ2" := "ContadorSimiJ2";
       "BloqueoSimilares6" := FALSE;
   END_IF;
   #_w32 := #_w25 AND "BloqueoSimilares7";
   IF #_w32 THEN "Var".CodigoSimilaresJ2[2] := 8; END_IF;
   "ContadorSimilaresJ2".CTU(CU := #_w32, R := "ReiniciarChecarSimiJ2", PV := 3, CV => "ContadorSimiJ2");
   IF #_w32 THEN
       "ContadorSimiTempJ2" := "ContadorSimiJ2";
       "BloqueoSimilares7" := FALSE;
   END_IF;
END_REGION

REGION Network 25: Amarillo J2
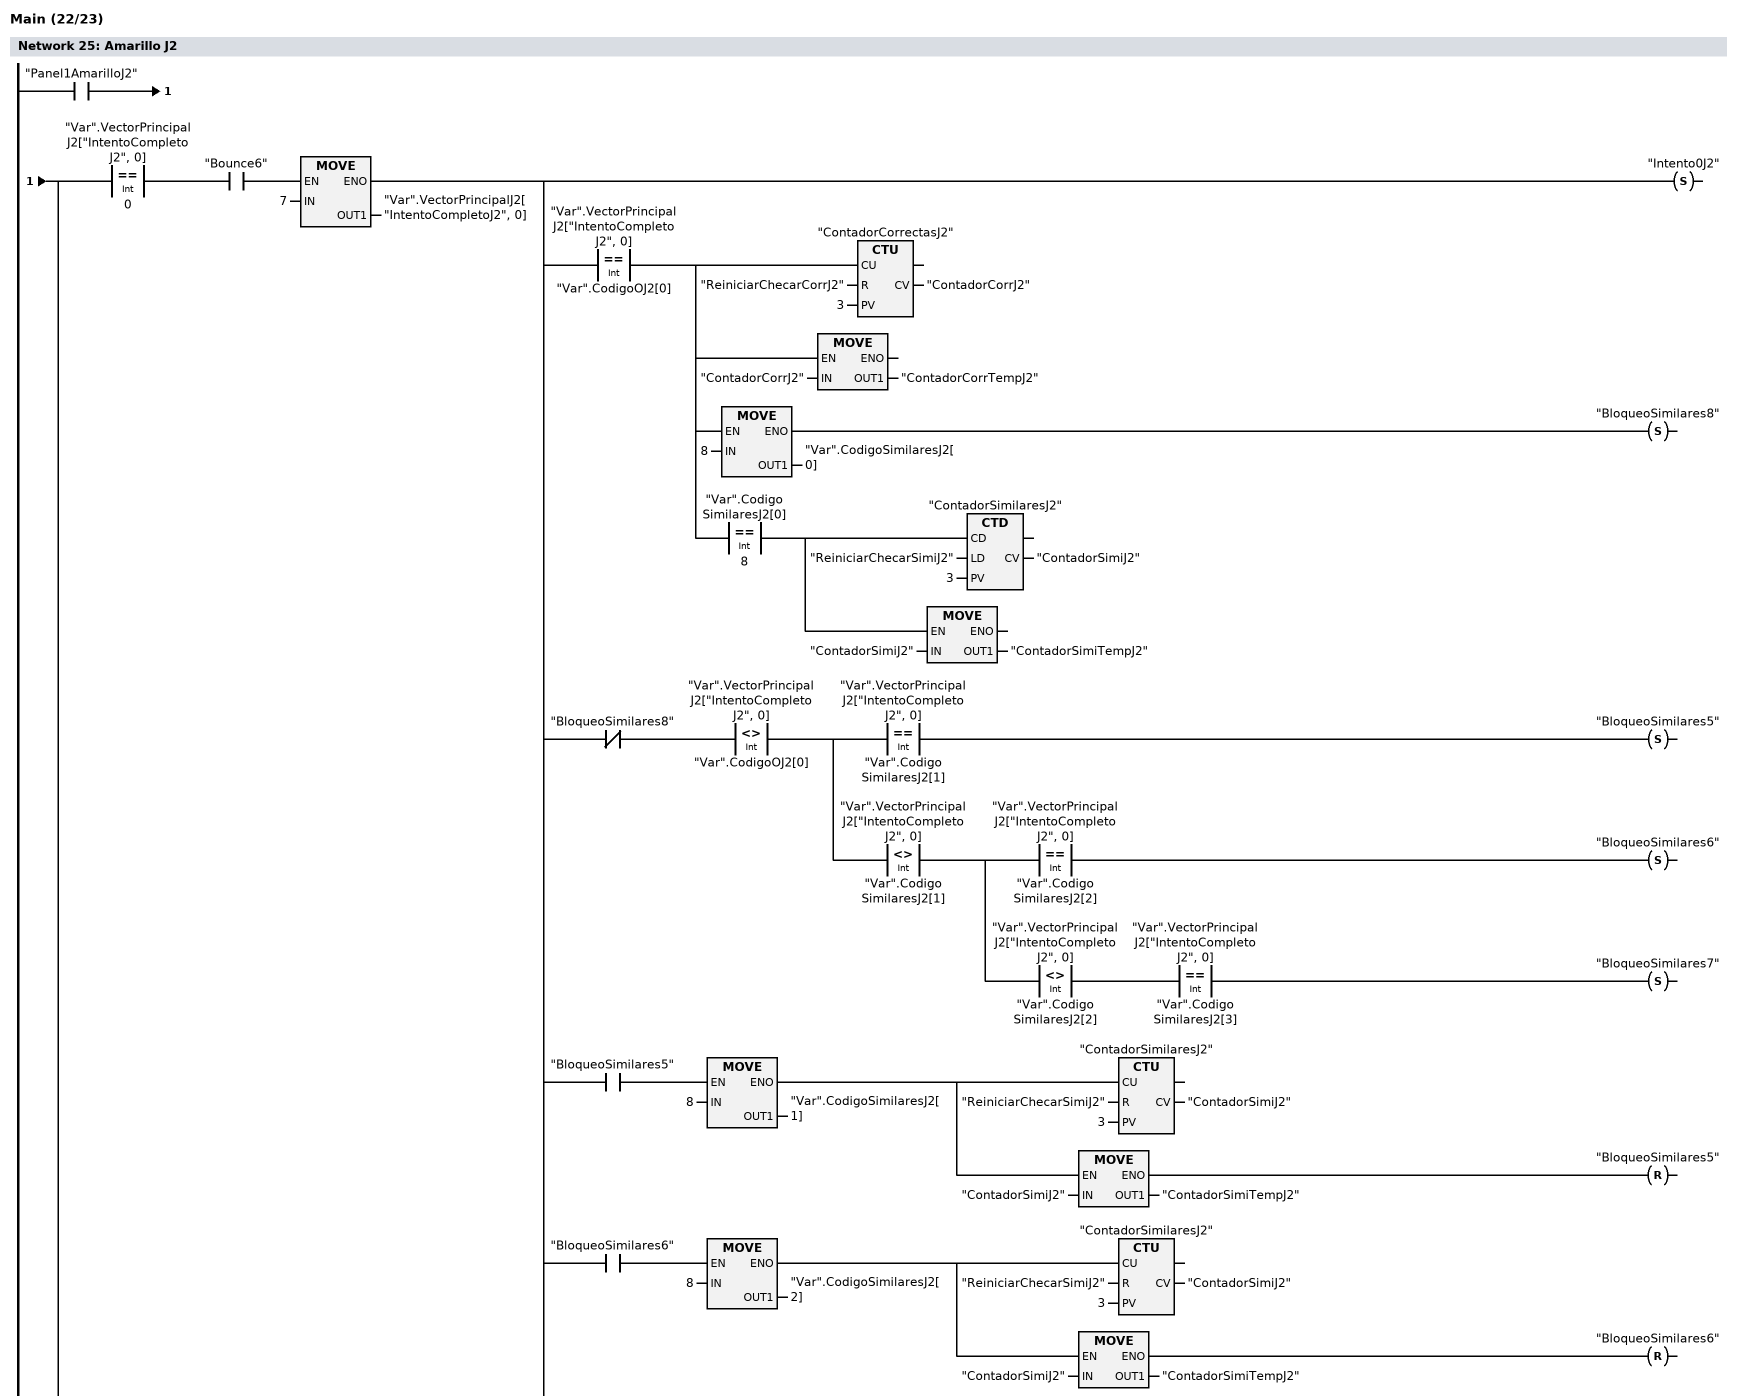
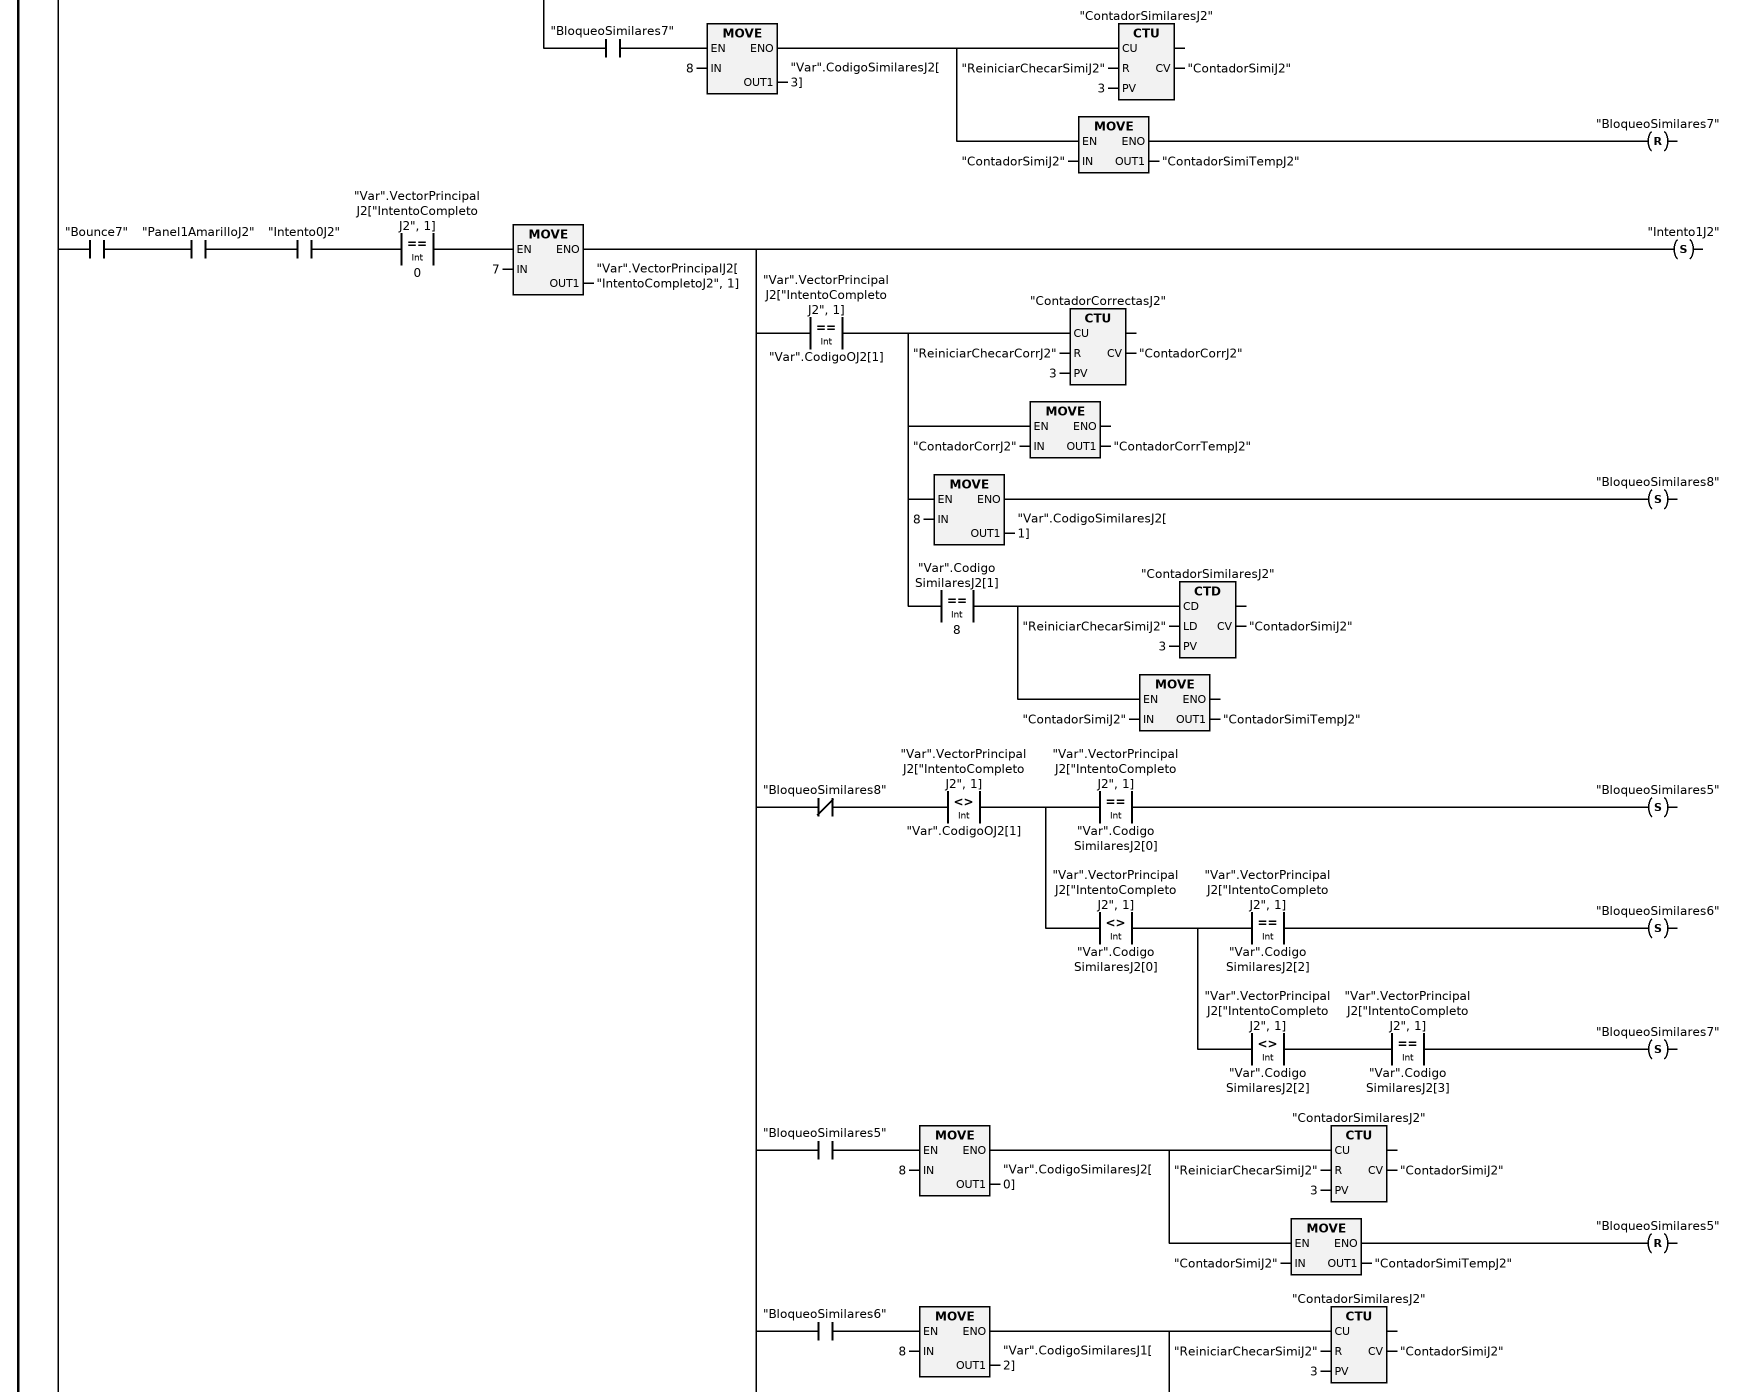
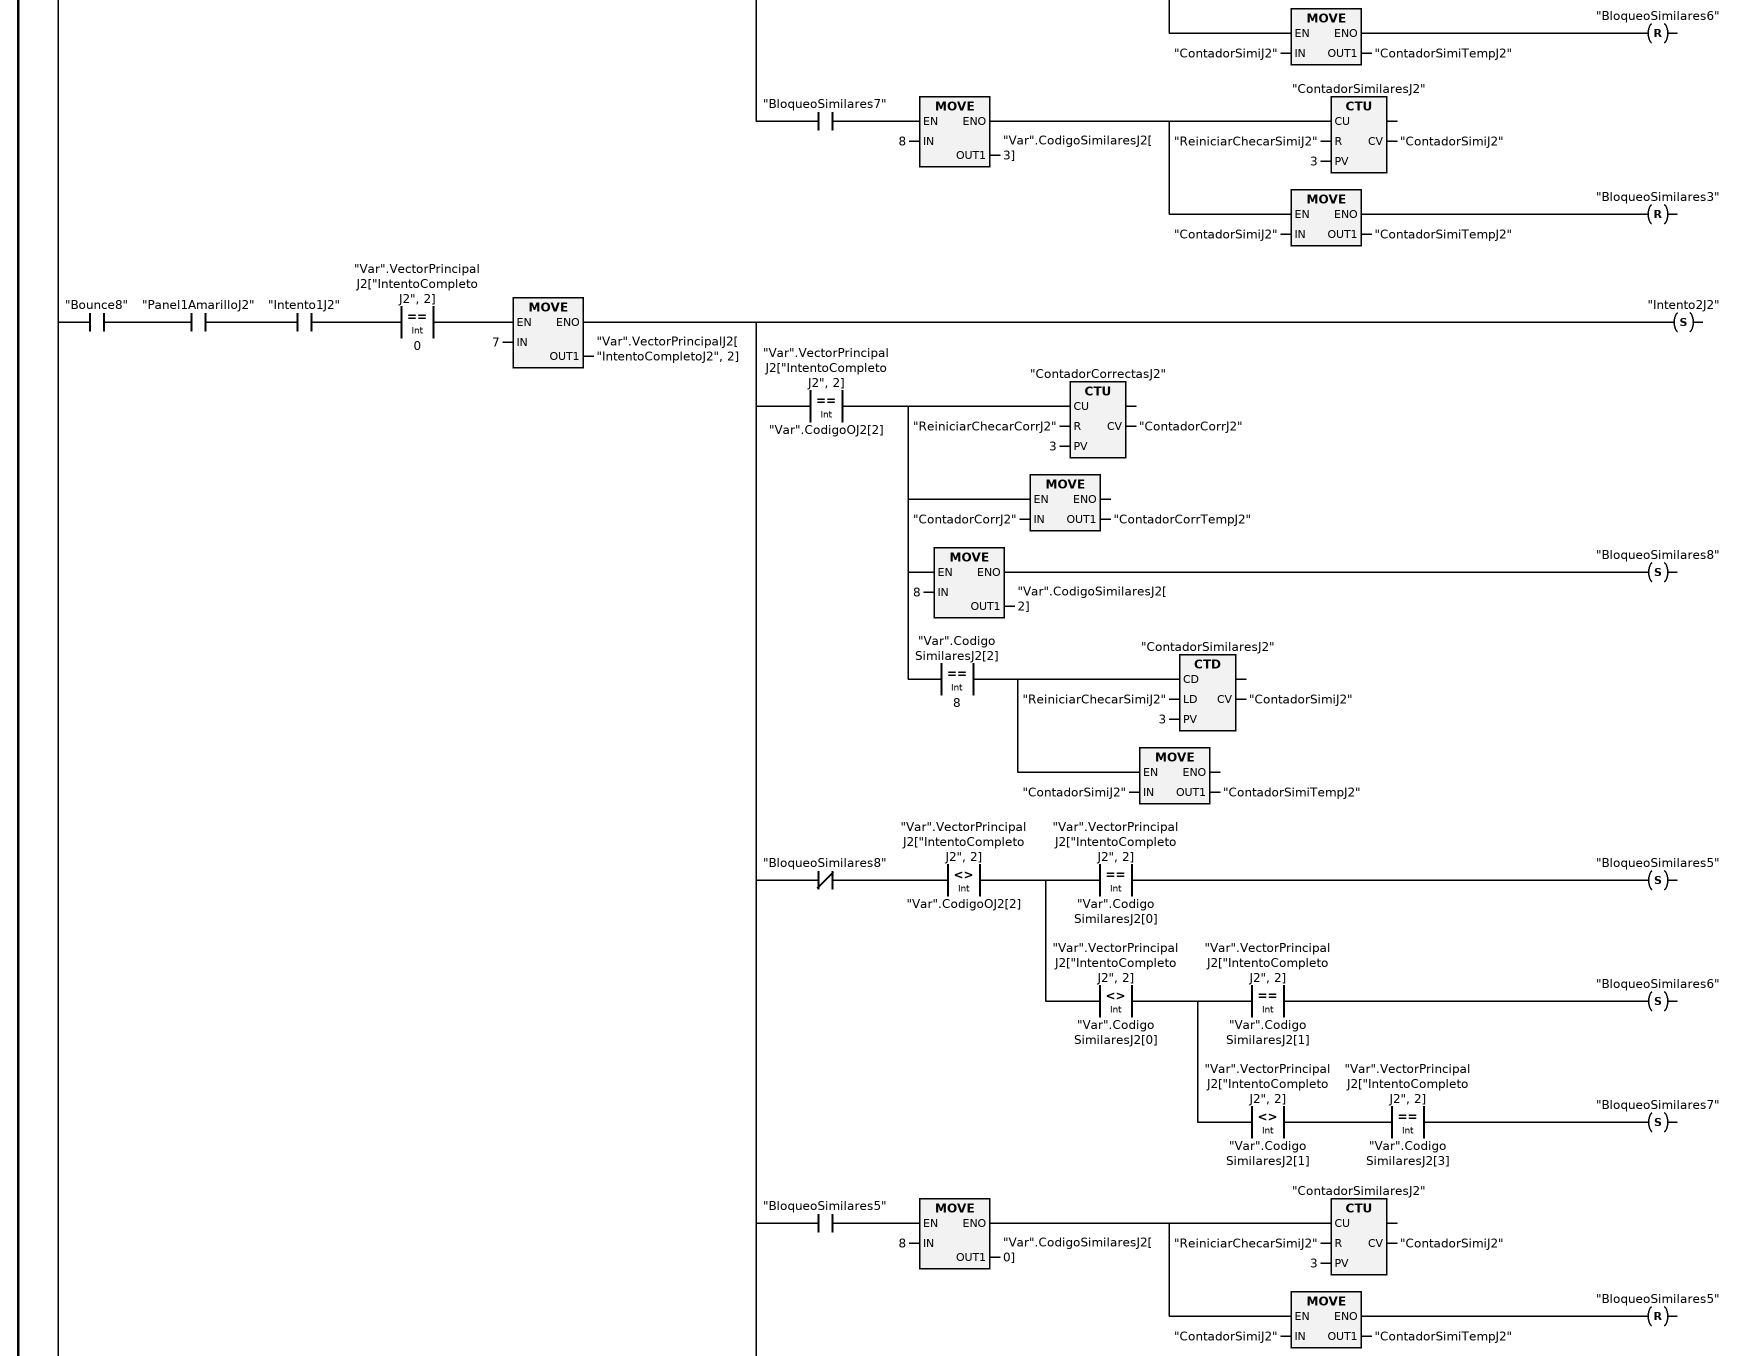
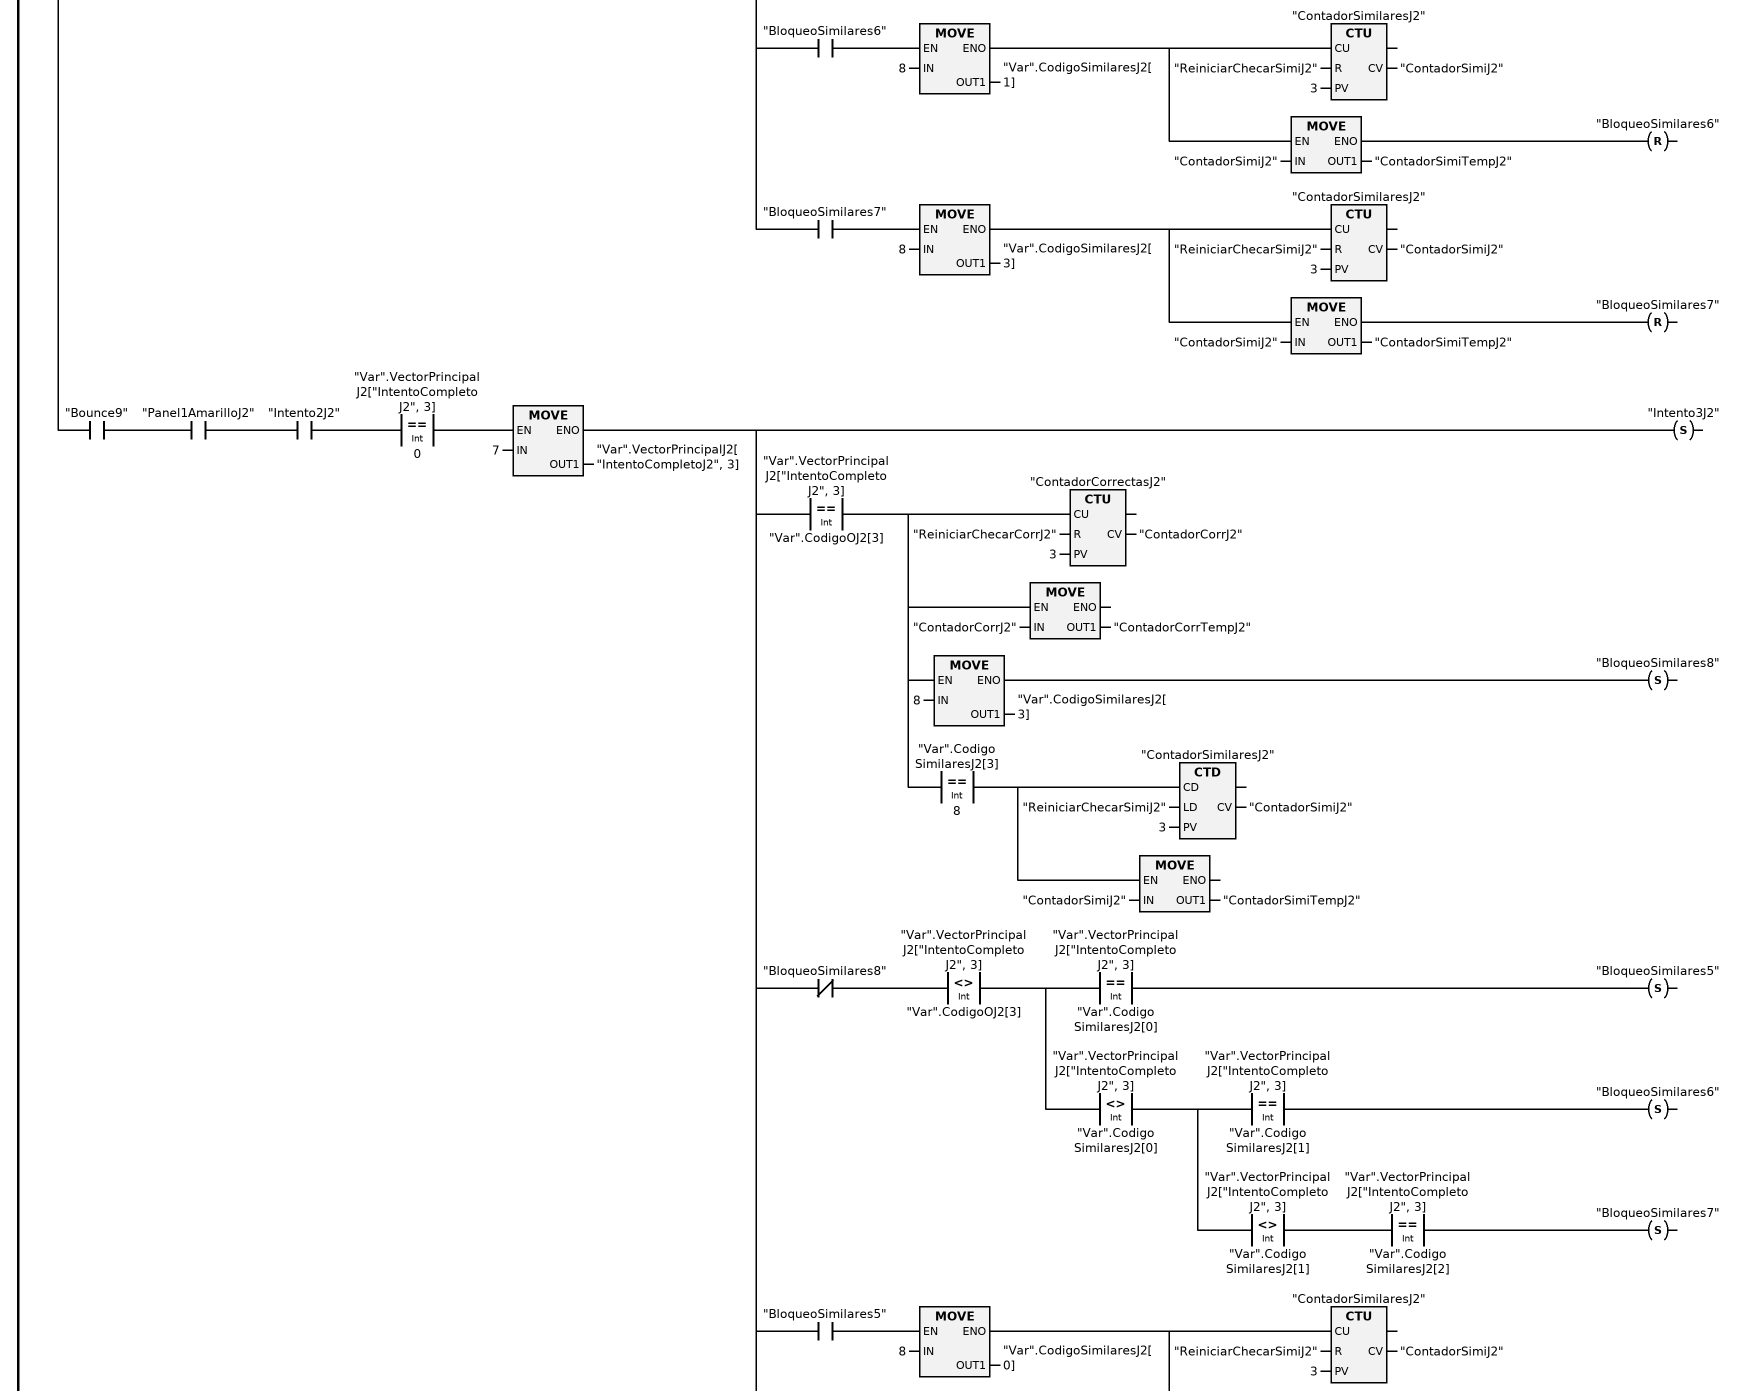
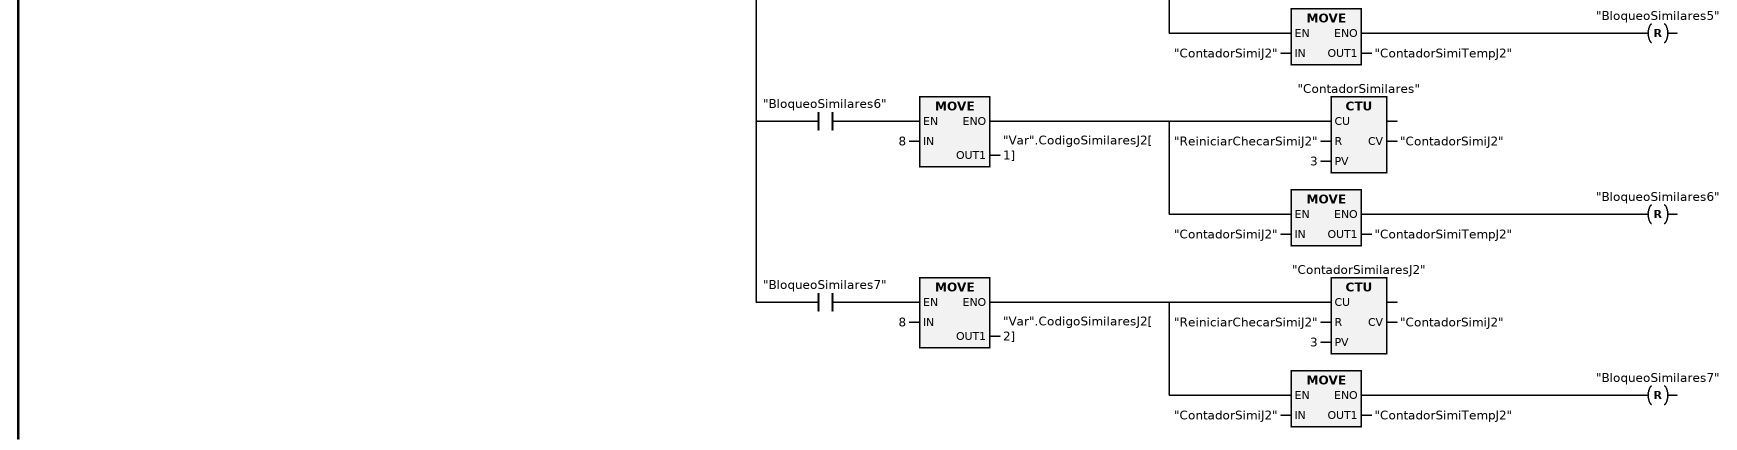
   #_w1 := "Panel1AmarilloJ2" AND ("Var".VectorPrincipalJ2["IntentoCompletoJ2", 0] = 0) AND "Bounce6";
   IF #_w1 THEN
       "Var".VectorPrincipalJ2["IntentoCompletoJ2", 0] := 7;
       "Intento0J2" := TRUE;
   END_IF;
   #_w2 := #_w1 AND ("Var".VectorPrincipalJ2["IntentoCompletoJ2", 0] = "Var".CodigoOJ2[0]);
   "ContadorCorrectasJ2".CTU(CU := #_w2, R := "ReiniciarChecarCorrJ2", PV := 3, CV => "ContadorCorrJ2");
   IF #_w2 THEN
       "ContadorCorrTempJ2" := "ContadorCorrJ2";
       "Var".CodigoSimilaresJ2[0] := 8;
       "BloqueoSimilares8" := TRUE;
   END_IF;
   #_w3 := #_w2 AND ("Var".CodigoSimilaresJ2[0] = 8);
   "ContadorSimilaresJ2".CTD(CD := #_w3, LD := "ReiniciarChecarSimiJ2", PV := 3, CV => "ContadorSimiJ2");
   IF #_w3 THEN "ContadorSimiTempJ2" := "ContadorSimiJ2"; END_IF;
   #_w4 := #_w1 AND NOT "BloqueoSimilares8" AND ("Var".VectorPrincipalJ2["IntentoCompletoJ2", 0] <> "Var".CodigoOJ2[0]);
   IF #_w4 AND ("Var".VectorPrincipalJ2["IntentoCompletoJ2", 0] = "Var".CodigoSimilaresJ2[1]) THEN
       "BloqueoSimilares5" := TRUE;
   END_IF;
   #_w5 := #_w4 AND ("Var".VectorPrincipalJ2["IntentoCompletoJ2", 0] <> "Var".CodigoSimilaresJ2[1]);
   IF #_w5 AND ("Var".VectorPrincipalJ2["IntentoCompletoJ2", 0] = "Var".CodigoSimilaresJ2[2]) THEN
       "BloqueoSimilares6" := TRUE;
   END_IF;
   IF #_w5 AND ("Var".VectorPrincipalJ2["IntentoCompletoJ2", 0] <> "Var".CodigoSimilaresJ2[2]) AND ("Var".VectorPrincipalJ2["IntentoCompletoJ2", 0] = "Var".CodigoSimilaresJ2[3]) THEN
       "BloqueoSimilares7" := TRUE;
   END_IF;
   #_w6 := #_w1 AND "BloqueoSimilares5";
   IF #_w6 THEN "Var".CodigoSimilaresJ2[1] := 8; END_IF;
   "ContadorSimilaresJ2".CTU(CU := #_w6, R := "ReiniciarChecarSimiJ2", PV := 3, CV => "ContadorSimiJ2");
   IF #_w6 THEN
       "ContadorSimiTempJ2" := "ContadorSimiJ2";
       "BloqueoSimilares5" := FALSE;
   END_IF;
   #_w7 := #_w1 AND "BloqueoSimilares6";
   IF #_w7 THEN "Var".CodigoSimilaresJ2[2] := 8; END_IF;
   "ContadorSimilaresJ2".CTU(CU := #_w7, R := "ReiniciarChecarSimiJ2", PV := 3, CV => "ContadorSimiJ2");
   IF #_w7 THEN
       "ContadorSimiTempJ2" := "ContadorSimiJ2";
       "BloqueoSimilares6" := FALSE;
   END_IF;
   #_w8 := #_w1 AND "BloqueoSimilares7";
   IF #_w8 THEN "Var".CodigoSimilaresJ2[3] := 8; END_IF;
   "ContadorSimilaresJ2".CTU(CU := #_w8, R := "ReiniciarChecarSimiJ2", PV := 3, CV => "ContadorSimiJ2");
   IF #_w8 THEN
       "ContadorSimiTempJ2" := "ContadorSimiJ2";
       "BloqueoSimilares7" := FALSE;
   END_IF;
   #_w9 := "Panel1AmarilloJ2" AND "Bounce7" AND "Panel1AmarilloJ2" AND "Intento0J2" AND ("Var".VectorPrincipalJ2["IntentoCompletoJ2", 1] = 0);
   IF #_w9 THEN
       "Var".VectorPrincipalJ2["IntentoCompletoJ2", 1] := 7;
       "Intento1J2" := TRUE;
   END_IF;
   #_w10 := #_w9 AND ("Var".VectorPrincipalJ2["IntentoCompletoJ2", 1] = "Var".CodigoOJ2[1]);
   "ContadorCorrectasJ2".CTU(CU := #_w10, R := "ReiniciarChecarCorrJ2", PV := 3, CV => "ContadorCorrJ2");
   IF #_w10 THEN
       "ContadorCorrTempJ2" := "ContadorCorrJ2";
       "Var".CodigoSimilaresJ2[1] := 8;
       "BloqueoSimilares8" := TRUE;
   END_IF;
   #_w11 := #_w10 AND ("Var".CodigoSimilaresJ2[1] = 8);
   "ContadorSimilaresJ2".CTD(CD := #_w11, LD := "ReiniciarChecarSimiJ2", PV := 3, CV => "ContadorSimiJ2");
   IF #_w11 THEN "ContadorSimiTempJ2" := "ContadorSimiJ2"; END_IF;
   #_w12 := #_w9 AND NOT "BloqueoSimilares8" AND ("Var".VectorPrincipalJ2["IntentoCompletoJ2", 1] <> "Var".CodigoOJ2[1]);
   IF #_w12 AND ("Var".VectorPrincipalJ2["IntentoCompletoJ2", 1] = "Var".CodigoSimilaresJ2[0]) THEN
       "BloqueoSimilares5" := TRUE;
   END_IF;
   #_w13 := #_w12 AND ("Var".VectorPrincipalJ2["IntentoCompletoJ2", 1] <> "Var".CodigoSimilaresJ2[0]);
   IF #_w13 AND ("Var".VectorPrincipalJ2["IntentoCompletoJ2", 1] = "Var".CodigoSimilaresJ2[2]) THEN
       "BloqueoSimilares6" := TRUE;
   END_IF;
   IF #_w13 AND ("Var".VectorPrincipalJ2["IntentoCompletoJ2", 1] <> "Var".CodigoSimilaresJ2[2]) AND ("Var".VectorPrincipalJ2["IntentoCompletoJ2", 1] = "Var".CodigoSimilaresJ2[3]) THEN
       "BloqueoSimilares7" := TRUE;
   END_IF;
   #_w14 := #_w9 AND "BloqueoSimilares5";
   IF #_w14 THEN "Var".CodigoSimilaresJ2[0] := 8; END_IF;
   "ContadorSimilaresJ2".CTU(CU := #_w14, R := "ReiniciarChecarSimiJ2", PV := 3, CV => "ContadorSimiJ2");
   IF #_w14 THEN
       "ContadorSimiTempJ2" := "ContadorSimiJ2";
       "BloqueoSimilares5" := FALSE;
   END_IF;
   #_w15 := #_w9 AND "BloqueoSimilares6";
   IF #_w15 THEN "Var".CodigoSimilaresJ1[2] := 8; END_IF;
   "ContadorSimilaresJ2".CTU(CU := #_w15, R := "ReiniciarChecarSimiJ2", PV := 3, CV => "ContadorSimiJ2");
   IF #_w15 THEN
       "ContadorSimiTempJ2" := "ContadorSimiJ2";
       "BloqueoSimilares6" := FALSE;
   END_IF;
   #_w16 := #_w9 AND "BloqueoSimilares7";
   IF #_w16 THEN "Var".CodigoSimilaresJ2[3] := 8; END_IF;
   "ContadorSimilaresJ2".CTU(CU := #_w16, R := "ReiniciarChecarSimiJ2", PV := 3, CV => "ContadorSimiJ2");
   IF #_w16 THEN
       "ContadorSimiTempJ2" := "ContadorSimiJ2";
       "BloqueoSimilares3" := FALSE;
   END_IF;
   #_w17 := "Panel1AmarilloJ2" AND "Bounce8" AND "Panel1AmarilloJ2" AND "Intento1J2" AND ("Var".VectorPrincipalJ2["IntentoCompletoJ2", 2] = 0);
   IF #_w17 THEN
       "Var".VectorPrincipalJ2["IntentoCompletoJ2", 2] := 7;
       "Intento2J2" := TRUE;
   END_IF;
   #_w18 := #_w17 AND ("Var".VectorPrincipalJ2["IntentoCompletoJ2", 2] = "Var".CodigoOJ2[2]);
   "ContadorCorrectasJ2".CTU(CU := #_w18, R := "ReiniciarChecarCorrJ2", PV := 3, CV => "ContadorCorrJ2");
   IF #_w18 THEN
       "ContadorCorrTempJ2" := "ContadorCorrJ2";
       "Var".CodigoSimilaresJ2[2] := 8;
       "BloqueoSimilares8" := TRUE;
   END_IF;
   #_w19 := #_w18 AND ("Var".CodigoSimilaresJ2[2] = 8);
   "ContadorSimilaresJ2".CTD(CD := #_w19, LD := "ReiniciarChecarSimiJ2", PV := 3, CV => "ContadorSimiJ2");
   IF #_w19 THEN "ContadorSimiTempJ2" := "ContadorSimiJ2"; END_IF;
   #_w20 := #_w17 AND NOT "BloqueoSimilares8" AND ("Var".VectorPrincipalJ2["IntentoCompletoJ2", 2] <> "Var".CodigoOJ2[2]);
   IF #_w20 AND ("Var".VectorPrincipalJ2["IntentoCompletoJ2", 2] = "Var".CodigoSimilaresJ2[0]) THEN
       "BloqueoSimilares5" := TRUE;
   END_IF;
   #_w21 := #_w20 AND ("Var".VectorPrincipalJ2["IntentoCompletoJ2", 2] <> "Var".CodigoSimilaresJ2[0]);
   IF #_w21 AND ("Var".VectorPrincipalJ2["IntentoCompletoJ2", 2] = "Var".CodigoSimilaresJ2[1]) THEN
       "BloqueoSimilares6" := TRUE;
   END_IF;
   IF #_w21 AND ("Var".VectorPrincipalJ2["IntentoCompletoJ2", 2] <> "Var".CodigoSimilaresJ2[1]) AND ("Var".VectorPrincipalJ2["IntentoCompletoJ2", 2] = "Var".CodigoSimilaresJ2[3]) THEN
       "BloqueoSimilares7" := TRUE;
   END_IF;
   #_w22 := #_w17 AND "BloqueoSimilares5";
   IF #_w22 THEN "Var".CodigoSimilaresJ2[0] := 8; END_IF;
   "ContadorSimilaresJ2".CTU(CU := #_w22, R := "ReiniciarChecarSimiJ2", PV := 3, CV => "ContadorSimiJ2");
   IF #_w22 THEN
       "ContadorSimiTempJ2" := "ContadorSimiJ2";
       "BloqueoSimilares5" := FALSE;
   END_IF;
   #_w23 := #_w17 AND "BloqueoSimilares6";
   IF #_w23 THEN "Var".CodigoSimilaresJ2[1] := 8; END_IF;
   "ContadorSimilaresJ2".CTU(CU := #_w23, R := "ReiniciarChecarSimiJ2", PV := 3, CV => "ContadorSimiJ2");
   IF #_w23 THEN
       "ContadorSimiTempJ2" := "ContadorSimiJ2";
       "BloqueoSimilares6" := FALSE;
   END_IF;
   #_w24 := #_w17 AND "BloqueoSimilares7";
   IF #_w24 THEN "Var".CodigoSimilaresJ2[3] := 8; END_IF;
   "ContadorSimilaresJ2".CTU(CU := #_w24, R := "ReiniciarChecarSimiJ2", PV := 3, CV => "ContadorSimiJ2");
   IF #_w24 THEN
       "ContadorSimiTempJ2" := "ContadorSimiJ2";
       "BloqueoSimilares7" := FALSE;
   END_IF;
   #_w25 := "Panel1AmarilloJ2" AND "Bounce9" AND "Panel1AmarilloJ2" AND "Intento2J2" AND ("Var".VectorPrincipalJ2["IntentoCompletoJ2", 3] = 0);
   IF #_w25 THEN
       "Var".VectorPrincipalJ2["IntentoCompletoJ2", 3] := 7;
       "Intento3J2" := TRUE;
   END_IF;
   #_w26 := #_w25 AND ("Var".VectorPrincipalJ2["IntentoCompletoJ2", 3] = "Var".CodigoOJ2[3]);
   "ContadorCorrectasJ2".CTU(CU := #_w26, R := "ReiniciarChecarCorrJ2", PV := 3, CV => "ContadorCorrJ2");
   IF #_w26 THEN
       "ContadorCorrTempJ2" := "ContadorCorrJ2";
       "Var".CodigoSimilaresJ2[3] := 8;
       "BloqueoSimilares8" := TRUE;
   END_IF;
   #_w27 := #_w26 AND ("Var".CodigoSimilaresJ2[3] = 8);
   "ContadorSimilaresJ2".CTD(CD := #_w27, LD := "ReiniciarChecarSimiJ2", PV := 3, CV => "ContadorSimiJ2");
   IF #_w27 THEN "ContadorSimiTempJ2" := "ContadorSimiJ2"; END_IF;
   #_w28 := #_w25 AND NOT "BloqueoSimilares8" AND ("Var".VectorPrincipalJ2["IntentoCompletoJ2", 3] <> "Var".CodigoOJ2[3]);
   IF #_w28 AND ("Var".VectorPrincipalJ2["IntentoCompletoJ2", 3] = "Var".CodigoSimilaresJ2[0]) THEN
       "BloqueoSimilares5" := TRUE;
   END_IF;
   #_w29 := #_w28 AND ("Var".VectorPrincipalJ2["IntentoCompletoJ2", 3] <> "Var".CodigoSimilaresJ2[0]);
   IF #_w29 AND ("Var".VectorPrincipalJ2["IntentoCompletoJ2", 3] = "Var".CodigoSimilaresJ2[1]) THEN
       "BloqueoSimilares6" := TRUE;
   END_IF;
   IF #_w29 AND ("Var".VectorPrincipalJ2["IntentoCompletoJ2", 3] <> "Var".CodigoSimilaresJ2[1]) AND ("Var".VectorPrincipalJ2["IntentoCompletoJ2", 3] = "Var".CodigoSimilaresJ2[2]) THEN
       "BloqueoSimilares7" := TRUE;
   END_IF;
   #_w30 := #_w25 AND "BloqueoSimilares5";
   IF #_w30 THEN "Var".CodigoSimilaresJ2[0] := 8; END_IF;
   "ContadorSimilaresJ2".CTU(CU := #_w30, R := "ReiniciarChecarSimiJ2", PV := 3, CV => "ContadorSimiJ2");
   IF #_w30 THEN
       "ContadorSimiTempJ2" := "ContadorSimiJ2";
       "BloqueoSimilares5" := FALSE;
   END_IF;
   #_w31 := #_w25 AND "BloqueoSimilares6";
   IF #_w31 THEN "Var".CodigoSimilaresJ2[1] := 8; END_IF;
   "ContadorSimilares".CTU(CU := #_w31, R := "ReiniciarChecarSimiJ2", PV := 3, CV => "ContadorSimiJ2");
   IF #_w31 THEN
       "ContadorSimiTempJ2" := "ContadorSimiJ2";
       "BloqueoSimilares6" := FALSE;
   END_IF;
   #_w32 := #_w25 AND "BloqueoSimilares7";
   IF #_w32 THEN "Var".CodigoSimilaresJ2[2] := 8; END_IF;
   "ContadorSimilaresJ2".CTU(CU := #_w32, R := "ReiniciarChecarSimiJ2", PV := 3, CV => "ContadorSimiJ2");
   IF #_w32 THEN
       "ContadorSimiTempJ2" := "ContadorSimiJ2";
       "BloqueoSimilares7" := FALSE;
   END_IF;
END_REGION

REGION Network 26: Comprobar Intentos J2
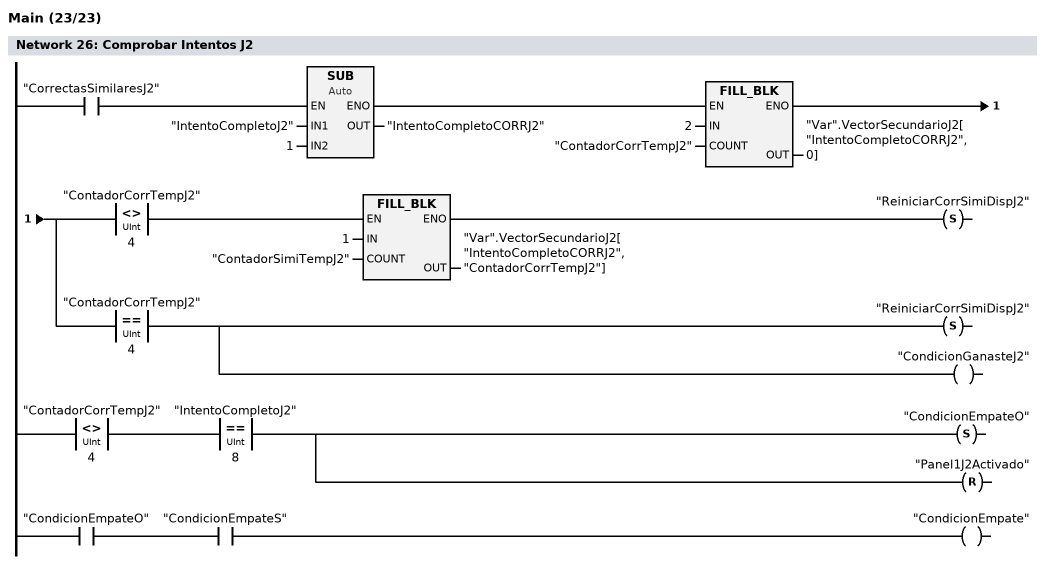
   RUNG wire#powerrail
      Contact( "CorrectasSimilaresJ2" )
      Sub(in1 := "IntentoCompletoJ2", in2 := 1, out => "IntentoCompletoCORRJ2")
      FillBlockI(in := 2, count := "ContadorCorrTempJ2", out => "Var".VectorSecundarioJ2["IntentoCompletoCORRJ2", 0])
      wire#w1
      { S7_Templates := "SrcType := UInt" } NE_Contact(in1 := "ContadorCorrTempJ2", in2 := 4)
      FillBlockI(in := 1, count := "ContadorSimiTempJ2", out => "Var".VectorSecundarioJ2["IntentoCompletoCORRJ2", "ContadorCorrTempJ2"])
      S_Coil( "ReiniciarCorrSimiDispJ2" )
   END_RUNG
   RUNG wire#w1
      { S7_Templates := "SrcType := UInt" } EQ_Contact(in1 := "ContadorCorrTempJ2", in2 := 4)
      wire#w2
      S_Coil( "ReiniciarCorrSimiDispJ2" )
   END_RUNG
   RUNG wire#w2
      Coil( "CondicionGanasteJ2" )
   END_RUNG
   RUNG wire#powerrail
      { S7_Templates := "SrcType := UInt" } NE_Contact(in1 := "ContadorCorrTempJ2", in2 := 4)
      { S7_Templates := "SrcType := UInt" } EQ_Contact(in1 := "IntentoCompletoJ2", in2 := 8)
      wire#w3
      S_Coil( "CondicionEmpateO" )
   END_RUNG
   RUNG wire#w3
      R_Coil( "Panel1J2Activado" )
   END_RUNG
   RUNG wire#powerrail
      Contact( "CondicionEmpateO" )
      Contact( "CondicionEmpateS" )
      Coil( "CondicionEmpate" )
   END_RUNG
   // the same network as SCL:
   IF "CorrectasSimilaresJ2" THEN "IntentoCompletoCORRJ2" := "IntentoCompletoJ2" - 1; END_IF;
   #_w1 := "CorrectasSimilaresJ2";
   IF #_w1 THEN
       FILL_BLK(IN := 2, COUNT := "ContadorCorrTempJ2", OUT => "Var".VectorSecundarioJ2["IntentoCompletoCORRJ2", 0]);
   END_IF;
   #_w2 := #_w1 AND ("ContadorCorrTempJ2" <> 4);
   IF #_w2 THEN
       FILL_BLK(IN := 1,
                COUNT := "ContadorSimiTempJ2",
                OUT => "Var".VectorSecundarioJ2["IntentoCompletoCORRJ2", "ContadorCorrTempJ2"]);
       "ReiniciarCorrSimiDispJ2" := TRUE;
   END_IF;
   #_w3 := #_w1 AND ("ContadorCorrTempJ2" = 4);
   IF #_w3 THEN "ReiniciarCorrSimiDispJ2" := TRUE; END_IF;
   "CondicionGanasteJ2" := #_w3;
   IF ("ContadorCorrTempJ2" <> 4) AND ("IntentoCompletoJ2" = 8) THEN
       "CondicionEmpateO" := TRUE;
       "Panel1J2Activado" := FALSE;
   END_IF;
   "CondicionEmpate" := "CondicionEmpateO" AND "CondicionEmpateS";
END_REGION
END_ORGANIZATION_BLOCK

(* ===== HMI "HMI_RT_1" =====
system functions are stored by id; their names below are inferred from use
connection "HMI_Connection_1": ETHERNET, S7_1500_OMS

HMI tags "Default tag table"
   "Tag_ScreenNumber" : UInt, internal
   "ReiniciarJuego" : Bool = PLC ReiniciarJuego AT %M6.0, 1 s
   "Panel2CafeJ1" : Bool = PLC Panel2CafeJ1 AT %M10.4, 1 s
   "Panel2RosaJ1" : Bool = PLC Panel2RosaJ1 AT %M10.5, 1 s
   "Panel2MoradoJ1" : Bool = PLC Panel2MoradoJ1 AT %M10.6, 1 s
   "Panel2RojoJ1" : Bool = PLC Panel2RojoJ1 AT %M10.7, 1 s
   "Panel2AzulJ1" : Bool = PLC Panel2AzulJ1 AT %M11.0, 1 s
   "Panel2VerdeJ1" : Bool = PLC Panel2VerdeJ1 AT %M11.1, 1 s
   "Panel2AmarilloJ1" : Bool = PLC Panel2AmarilloJ1 AT %M11.2, 1 s
   "Panel1CafeJ1" : Bool = PLC Panel1CafeJ1 AT %M9.5, 1 s
   "Panel1RosaJ1" : Bool = PLC Panel1RosaJ1 AT %M9.6, 1 s
   "Panel1MoradoJ1" : Bool = PLC Panel1MoradoJ1 AT %M9.7, 1 s
   "Panel1RojoJ1" : Bool = PLC Panel1RojoJ1 AT %M10.0, 1 s
   "Panel1AzulJ1" : Bool = PLC Panel1AzulJ1 AT %M10.1, 1 s
   "Panel1VerdeJ1" : Bool = PLC Panel1VerdeJ1 AT %M10.2, 1 s
   "Panel1AmarilloJ1" : Bool = PLC Panel1AmarilloJ1 AT %M10.3, 1 s
   "Panel1J1Activado" : Bool = PLC Panel1J1Activado AT %M13.1, 1 s
   "Panel2J1Activado" : Bool = PLC Panel2J1Activado AT %M13.2, 1 s
   "Var_VectorMensajes{0}" : Int = PLC "Var".VectorMensajes[0], 1 s
   "Var_VectorMensajes{1}" : Int = PLC "Var".VectorMensajes[1], 1 s
   "Var_VectorMensajes{2}" : Int = PLC "Var".VectorMensajes[2], 1 s
   "Var_VectorMensajes{3}" : Int = PLC "Var".VectorMensajes[3], 1 s
   "Var_VectorMensajes{4}" : Int = PLC "Var".VectorMensajes[4], 1 s
   "Var_VectorMensajes{5}" : Int = PLC "Var".VectorMensajes[5], 1 s
   "Var_VectorMensajes{6}" : Int = PLC "Var".VectorMensajes[6], 1 s
   "Var_VectorMensajes{7}" : Int = PLC "Var".VectorMensajes[7], 1 s
   "Var_VectorMensajes{8}" : Int = PLC "Var".VectorMensajes[8], 1 s
   "Var_VectorMensajes{9}" : Int = PLC "Var".VectorMensajes[9], 1 s
   "Var_VectorMensajes{10}" : Int = PLC "Var".VectorMensajes[10], 1 s
   "Var_CodigoOJ1{0}" : Int = PLC "Var".CodigoOJ1[0], 1 s
   "Var_CodigoOJ1{1}" : Int = PLC "Var".CodigoOJ1[1], 1 s
   "Var_CodigoOJ1{2}" : Int = PLC "Var".CodigoOJ1[2], 1 s
   "Var_CodigoOJ1{3}" : Int = PLC "Var".CodigoOJ1[3], 1 s
   "Var_CodigoSJ1{0}" : Int = PLC "Var".CodigoSJ1[0], 1 s
   "Var_CodigoSJ1{1}" : Int = PLC "Var".CodigoSJ1[1], 1 s
   "Var_CodigoSJ1{2}" : Int = PLC "Var".CodigoSJ1[2], 1 s
   "Var_CodigoSJ1{3}" : Int = PLC "Var".CodigoSJ1[3], 1 s
   "Var_VectorPrincipalJ1{0,0}" : Int = PLC "Var".VectorPrincipalJ1[0,0], 1 s
   "Var_VectorPrincipalJ1{0,1}" : Int = PLC "Var".VectorPrincipalJ1[0,1], 1 s
   "Var_VectorPrincipalJ1{0,2}" : Int = PLC "Var".VectorPrincipalJ1[0,2], 1 s
   "Var_VectorPrincipalJ1{0,3}" : Int = PLC "Var".VectorPrincipalJ1[0,3], 1 s
   "Var_VectorPrincipalJ1{1,0}" : Int = PLC "Var".VectorPrincipalJ1[1,0], 1 s
   "Var_VectorPrincipalJ1{1,1}" : Int = PLC "Var".VectorPrincipalJ1[1,1], 1 s
   "Var_VectorPrincipalJ1{1,2}" : Int = PLC "Var".VectorPrincipalJ1[1,2], 1 s
   "Var_VectorPrincipalJ1{1,3}" : Int = PLC "Var".VectorPrincipalJ1[1,3], 1 s
   "Var_VectorPrincipalJ1{2,0}" : Int = PLC "Var".VectorPrincipalJ1[2,0], 1 s
   "Var_VectorPrincipalJ1{2,1}" : Int = PLC "Var".VectorPrincipalJ1[2,1], 1 s
   "Var_VectorPrincipalJ1{2,2}" : Int = PLC "Var".VectorPrincipalJ1[2,2], 1 s
   "Var_VectorPrincipalJ1{2,3}" : Int = PLC "Var".VectorPrincipalJ1[2,3], 1 s
   "Var_VectorPrincipalJ1{3,0}" : Int = PLC "Var".VectorPrincipalJ1[3,0], 1 s
   "Var_VectorPrincipalJ1{3,1}" : Int = PLC "Var".VectorPrincipalJ1[3,1], 1 s
   "Var_VectorPrincipalJ1{3,2}" : Int = PLC "Var".VectorPrincipalJ1[3,2], 1 s
   "Var_VectorPrincipalJ1{3,3}" : Int = PLC "Var".VectorPrincipalJ1[3,3], 1 s
   "Var_VectorPrincipalJ1{4,0}" : Int = PLC "Var".VectorPrincipalJ1[4,0], 1 s
   "Var_VectorPrincipalJ1{4,1}" : Int = PLC "Var".VectorPrincipalJ1[4,1], 1 s
   "Var_VectorPrincipalJ1{4,2}" : Int = PLC "Var".VectorPrincipalJ1[4,2], 1 s
   "Var_VectorPrincipalJ1{4,3}" : Int = PLC "Var".VectorPrincipalJ1[4,3], 1 s
   "Var_VectorPrincipalJ1{5,0}" : Int = PLC "Var".VectorPrincipalJ1[5,0], 1 s
   "Var_VectorPrincipalJ1{5,1}" : Int = PLC "Var".VectorPrincipalJ1[5,1], 1 s
   "Var_VectorPrincipalJ1{5,2}" : Int = PLC "Var".VectorPrincipalJ1[5,2], 1 s
   "Var_VectorPrincipalJ1{5,3}" : Int = PLC "Var".VectorPrincipalJ1[5,3], 1 s
   "Var_VectorPrincipalJ1{6,0}" : Int = PLC "Var".VectorPrincipalJ1[6,0], 1 s
   "Var_VectorPrincipalJ1{6,1}" : Int = PLC "Var".VectorPrincipalJ1[6,1], 1 s
   "Var_VectorPrincipalJ1{6,2}" : Int = PLC "Var".VectorPrincipalJ1[6,2], 1 s
   "Var_VectorPrincipalJ1{6,3}" : Int = PLC "Var".VectorPrincipalJ1[6,3], 1 s
   "Var_VectorPrincipalJ1{7,0}" : Int = PLC "Var".VectorPrincipalJ1[7,0], 1 s
   "Var_VectorPrincipalJ1{7,1}" : Int = PLC "Var".VectorPrincipalJ1[7,1], 1 s
   "Var_VectorPrincipalJ1{7,2}" : Int = PLC "Var".VectorPrincipalJ1[7,2], 1 s
   "Var_VectorPrincipalJ1{7,3}" : Int = PLC "Var".VectorPrincipalJ1[7,3], 1 s
   "Var_VectorSecundarioJ1{0,0}" : Int = PLC "Var".VectorSecundarioJ1[0,0], 1 s
   "Var_VectorSecundarioJ1{0,1}" : Int = PLC "Var".VectorSecundarioJ1[0,1], 1 s
   "Var_VectorSecundarioJ1{0,2}" : Int = PLC "Var".VectorSecundarioJ1[0,2], 1 s
   "Var_VectorSecundarioJ1{0,3}" : Int = PLC "Var".VectorSecundarioJ1[0,3], 1 s
   "Var_VectorSecundarioJ1{1,0}" : Int = PLC "Var".VectorSecundarioJ1[1,0], 1 s
   "Var_VectorSecundarioJ1{1,1}" : Int = PLC "Var".VectorSecundarioJ1[1,1], 1 s
   "Var_VectorSecundarioJ1{1,2}" : Int = PLC "Var".VectorSecundarioJ1[1,2], 1 s
   "Var_VectorSecundarioJ1{1,3}" : Int = PLC "Var".VectorSecundarioJ1[1,3], 1 s
   "Var_VectorSecundarioJ1{2,0}" : Int = PLC "Var".VectorSecundarioJ1[2,0], 1 s
   "Var_VectorSecundarioJ1{2,1}" : Int = PLC "Var".VectorSecundarioJ1[2,1], 1 s
   "Var_VectorSecundarioJ1{2,2}" : Int = PLC "Var".VectorSecundarioJ1[2,2], 1 s
   "Var_VectorSecundarioJ1{2,3}" : Int = PLC "Var".VectorSecundarioJ1[2,3], 1 s
   "Var_VectorSecundarioJ1{3,0}" : Int = PLC "Var".VectorSecundarioJ1[3,0], 1 s
   "Var_VectorSecundarioJ1{3,1}" : Int = PLC "Var".VectorSecundarioJ1[3,1], 1 s
   "Var_VectorSecundarioJ1{3,2}" : Int = PLC "Var".VectorSecundarioJ1[3,2], 1 s
   "Var_VectorSecundarioJ1{3,3}" : Int = PLC "Var".VectorSecundarioJ1[3,3], 1 s
   "Var_VectorSecundarioJ1{4,0}" : Int = PLC "Var".VectorSecundarioJ1[4,0], 1 s
   "Var_VectorSecundarioJ1{4,1}" : Int = PLC "Var".VectorSecundarioJ1[4,1], 1 s
   "Var_VectorSecundarioJ1{4,2}" : Int = PLC "Var".VectorSecundarioJ1[4,2], 1 s
   "Var_VectorSecundarioJ1{4,3}" : Int = PLC "Var".VectorSecundarioJ1[4,3], 1 s
   "Var_VectorSecundarioJ1{5,0}" : Int = PLC "Var".VectorSecundarioJ1[5,0], 1 s
   "Var_VectorSecundarioJ1{5,1}" : Int = PLC "Var".VectorSecundarioJ1[5,1], 1 s
   "Var_VectorSecundarioJ1{5,2}" : Int = PLC "Var".VectorSecundarioJ1[5,2], 1 s
   "Var_VectorSecundarioJ1{5,3}" : Int = PLC "Var".VectorSecundarioJ1[5,3], 1 s
   "Var_VectorSecundarioJ1{6,0}" : Int = PLC "Var".VectorSecundarioJ1[6,0], 1 s
   "Var_VectorSecundarioJ1{6,1}" : Int = PLC "Var".VectorSecundarioJ1[6,1], 1 s
   "Var_VectorSecundarioJ1{6,2}" : Int = PLC "Var".VectorSecundarioJ1[6,2], 1 s
   "Var_VectorSecundarioJ1{6,3}" : Int = PLC "Var".VectorSecundarioJ1[6,3], 1 s
   "Var_VectorSecundarioJ1{7,0}" : Int = PLC "Var".VectorSecundarioJ1[7,0], 1 s
   "Var_VectorSecundarioJ1{7,1}" : Int = PLC "Var".VectorSecundarioJ1[7,1], 1 s
   "Var_VectorSecundarioJ1{7,2}" : Int = PLC "Var".VectorSecundarioJ1[7,2], 1 s
   "Var_VectorSecundarioJ1{7,3}" : Int = PLC "Var".VectorSecundarioJ1[7,3], 1 s
   "Bounce1" : Bool = PLC Bounce1 AT %M13.6, 1 s
   "Bounce5" : Bool = PLC Bounce5 AT %M14.1, 1 s
   "ReiniciarCorrSimiDisp" : Bool = PLC ReiniciarCorrSimiDisp AT %M34.0, 1 s
   "DescubrirCodigoSecreto" : Bool = PLC DescubrirCodigoSecreto AT %M50.3, 1 s

screen "Root screen" 800x442, template "Template_1"
   on GenerateScreen: SetTag("Tag_ScreenNumber", 1)
   Button "Button_3" at 67,293 size 28x26; TextOff 'Text'
      on Press: SetBit("Panel1CafeJ1")
      on Release: SetBit("Bounce5"); ResetBit("Panel1CafeJ1")
      Appearance <- "Panel1J1Activado"
   Button "Button_4" at 99,293 size 27x26; TextOff 'Text'
      on Press: SetBit("Panel1RosaJ1")
      on Release: SetBit("Bounce5"); ResetBit("Panel1RosaJ1")
      Appearance <- "Panel1J1Activado"
   Button "Button_5" at 131,293 size 27x24; TextOff 'Text'
      on Press: SetBit("Panel1MoradoJ1")
      on Release: SetBit("Bounce5"); ResetBit("Panel1MoradoJ1")
      Appearance <- "Panel1J1Activado"
   Button "Button_6" at 165,293 size 25x25; TextOff 'Text'
      on Press: SetBit("Panel1RojoJ1")
      on Release: SetBit("Bounce5"); ResetBit("Panel1RojoJ1")
      Appearance <- "Panel1J1Activado"
   Button "Button_7" at 196,293 size 25x24; TextOff 'Text'
      on Press: SetBit("Panel1AzulJ1")
      on Release: SetBit("Bounce5"); ResetBit("Panel1AzulJ1")
      Appearance <- "Panel1J1Activado"
   Button "Button_8" at 227,293 size 25x25; TextOff 'Text'
      on Press: SetBit("Panel1VerdeJ1")
      on Release: SetBit("Bounce5"); ResetBit("Panel1VerdeJ1")
      Appearance <- "Panel1J1Activado"
   Button "Button_9" at 256,294 size 25x23; TextOff 'Text'
      on Press: SetBit("Panel1AmarilloJ1")
      on Release: SetBit("Bounce5"); ResetBit("Panel1AmarilloJ1")
      Appearance <- "Panel1J1Activado"
   TextField "Text field_1" at 37,250 size 16x23; Text '1'
   TextField "Text field_2" at 37,221 size 16x23; Text '2'
   TextField "Text field_3" at 37,194 size 16x23; Text '3'
   TextField "Text field_4" at 37,163 size 16x23; Text '4'
   TextField "Text field_5" at 37,134 size 16x23; Text '5'
   TextField "Text field_6" at 37,103 size 16x23; Text '6'
   TextField "Text field_7" at 37,74 size 16x23; Text '7'
   TextField "Text field_8" at 37,43 size 16x23; Text '8'
   Circle "Circle_1" at 92,254 size 23x23
      Appearance <- "Var_VectorPrincipalJ1{0,0}"
   Circle "Circle_2" at 128,254 size 23x23
      Appearance <- "Var_VectorPrincipalJ1{0,1}"
   Circle "Circle_3" at 164,254 size 23x23
      Appearance <- "Var_VectorPrincipalJ1{0,2}"
   Circle "Circle_4" at 201,254 size 23x23
      Appearance <- "Var_VectorPrincipalJ1{0,3}"
   Circle "Circle_5" at 92,224 size 23x23
      Appearance <- "Var_VectorPrincipalJ1{1,0}"
   Circle "Circle_6" at 128,224 size 23x23
      Appearance <- "Var_VectorPrincipalJ1{1,1}"
   Circle "Circle_7" at 164,224 size 23x23
      Appearance <- "Var_VectorPrincipalJ1{1,2}"
   Circle "Circle_8" at 201,224 size 23x23
      Appearance <- "Var_VectorPrincipalJ1{1,3}"
   Circle "Circle_9" at 92,194 size 23x23
      Appearance <- "Var_VectorPrincipalJ1{2,0}"
   Circle "Circle_10" at 128,194 size 23x23
      Appearance <- "Var_VectorPrincipalJ1{2,1}"
   Circle "Circle_11" at 164,194 size 23x23
      Appearance <- "Var_VectorPrincipalJ1{2,2}"
   Circle "Circle_12" at 201,194 size 23x23
      Appearance <- "Var_VectorPrincipalJ1{2,3}"
   Circle "Circle_13" at 92,164 size 23x23
      Appearance <- "Var_VectorPrincipalJ1{3,0}"
   Circle "Circle_14" at 128,164 size 23x23
      Appearance <- "Var_VectorPrincipalJ1{3,1}"
   Circle "Circle_15" at 164,164 size 23x23
      Appearance <- "Var_VectorPrincipalJ1{3,2}"
   Circle "Circle_16" at 201,164 size 23x23
      Appearance <- "Var_VectorPrincipalJ1{3,3}"
   Circle "Circle_17" at 92,134 size 23x23
      Appearance <- "Var_VectorPrincipalJ1{4,0}"
   Circle "Circle_18" at 128,134 size 23x23
      Appearance <- "Var_VectorPrincipalJ1{4,1}"
   Circle "Circle_19" at 164,134 size 23x23
      Appearance <- "Var_VectorPrincipalJ1{4,2}"
   Circle "Circle_20" at 201,134 size 23x23
      Appearance <- "Var_VectorPrincipalJ1{4,3}"
   Circle "Circle_21" at 92,104 size 23x23
      Appearance <- "Var_VectorPrincipalJ1{5,0}"
   Circle "Circle_22" at 128,104 size 23x23
      Appearance <- "Var_VectorPrincipalJ1{5,1}"
   Circle "Circle_23" at 164,104 size 23x23
      Appearance <- "Var_VectorPrincipalJ1{5,2}"
   Circle "Circle_24" at 201,104 size 23x23
      Appearance <- "Var_VectorPrincipalJ1{5,3}"
   Circle "Circle_25" at 92,74 size 23x23
      Appearance <- "Var_VectorPrincipalJ1{6,0}"
   Circle "Circle_26" at 128,74 size 23x23
      Appearance <- "Var_VectorPrincipalJ1{6,1}"
   Circle "Circle_27" at 164,74 size 23x23
      Appearance <- "Var_VectorPrincipalJ1{6,2}"
   Circle "Circle_28" at 201,74 size 23x23
      Appearance <- "Var_VectorPrincipalJ1{6,3}"
   Circle "Circle_29" at 92,44 size 23x23
      Appearance <- "Var_VectorPrincipalJ1{7,0}"
   Circle "Circle_30" at 128,44 size 23x23
      Appearance <- "Var_VectorPrincipalJ1{7,1}"
   Circle "Circle_31" at 164,44 size 23x23
      Appearance <- "Var_VectorPrincipalJ1{7,2}"
   Circle "Circle_32" at 201,44 size 23x23
      Appearance <- "Var_VectorPrincipalJ1{7,3}"
   Circle "Circle_33" at 255,253 size 14x14
      Appearance <- "Var_VectorSecundarioJ1{0,0}"
   Circle "Circle_34" at 270,253 size 14x14
      Appearance <- "Var_VectorSecundarioJ1{0,1}"
   Circle "Circle_35" at 255,267 size 14x14
      Appearance <- "Var_VectorSecundarioJ1{0,2}"
   Circle "Circle_36" at 270,267 size 14x14
      Appearance <- "Var_VectorSecundarioJ1{0,3}"
   Circle "Circle_37" at 255,223 size 14x14
      Appearance <- "Var_VectorSecundarioJ1{1,0}"
   Circle "Circle_38" at 270,223 size 14x14
      Appearance <- "Var_VectorSecundarioJ1{1,1}"
   Circle "Circle_39" at 255,237 size 14x14
      Appearance <- "Var_VectorSecundarioJ1{1,2}"
   Circle "Circle_40" at 270,237 size 14x14
      Appearance <- "Var_VectorSecundarioJ1{1,3}"
   Circle "Circle_41" at 255,193 size 14x14
      Appearance <- "Var_VectorSecundarioJ1{2,0}"
   Circle "Circle_42" at 270,193 size 14x14
      Appearance <- "Var_VectorSecundarioJ1{2,1}"
   Circle "Circle_43" at 255,207 size 14x14
      Appearance <- "Var_VectorSecundarioJ1{2,2}"
   Circle "Circle_44" at 270,207 size 14x14
      Appearance <- "Var_VectorSecundarioJ1{2,3}"
   Circle "Circle_45" at 255,163 size 14x14
      Appearance <- "Var_VectorSecundarioJ1{3,0}"
   Circle "Circle_46" at 270,163 size 14x14
      Appearance <- "Var_VectorSecundarioJ1{3,1}"
   Circle "Circle_47" at 255,177 size 14x14
      Appearance <- "Var_VectorSecundarioJ1{3,2}"
   Circle "Circle_48" at 270,177 size 14x14
      Appearance <- "Var_VectorSecundarioJ1{3,3}"
   Circle "Circle_49" at 255,133 size 14x14
      Appearance <- "Var_VectorSecundarioJ1{4,0}"
   Circle "Circle_50" at 270,133 size 14x14
      Appearance <- "Var_VectorSecundarioJ1{4,1}"
   Circle "Circle_51" at 255,147 size 14x14
      Appearance <- "Var_VectorSecundarioJ1{4,2}"
   Circle "Circle_52" at 270,147 size 14x14
      Appearance <- "Var_VectorSecundarioJ1{4,3}"
   Circle "Circle_53" at 255,103 size 14x14
      Appearance <- "Var_VectorSecundarioJ1{5,0}"
   Circle "Circle_54" at 270,103 size 14x14
      Appearance <- "Var_VectorSecundarioJ1{5,1}"
   Circle "Circle_55" at 255,117 size 14x14
      Appearance <- "Var_VectorSecundarioJ1{5,2}"
   Circle "Circle_56" at 270,117 size 14x14
      Appearance <- "Var_VectorSecundarioJ1{5,3}"
   Circle "Circle_57" at 255,73 size 14x14
      Appearance <- "Var_VectorSecundarioJ1{6,0}"
   Circle "Circle_58" at 270,73 size 14x14
      Appearance <- "Var_VectorSecundarioJ1{6,1}"
   Circle "Circle_59" at 255,87 size 14x14
      Appearance <- "Var_VectorSecundarioJ1{6,2}"
   Circle "Circle_60" at 270,87 size 14x14
      Appearance <- "Var_VectorSecundarioJ1{6,3}"
   Circle "Circle_61" at 255,43 size 14x14
      Appearance <- "Var_VectorSecundarioJ1{7,0}"
   Circle "Circle_62" at 270,43 size 14x14
      Appearance <- "Var_VectorSecundarioJ1{7,1}"
   Circle "Circle_63" at 255,57 size 14x14
      Appearance <- "Var_VectorSecundarioJ1{7,2}"
   Circle "Circle_64" at 270,57 size 14x14
      Appearance <- "Var_VectorSecundarioJ1{7,3}"
   TextField "Text field_9" at 339,40 size 252x42; Text 'Selecciona el Codigo de tu Oponente:'
   TextField "Text field_10" at 383,22 size 162x23; Text 'INICIO Jugador 1'
   Circle "Circle_65" at 393,108 size 29x29
      Appearance <- "Var_CodigoSJ1{0}"
   Circle "Circle_66" at 431,107 size 29x29
      Appearance <- "Var_CodigoSJ1{1}"
   Circle "Circle_67" at 467,108 size 29x29
      Appearance <- "Var_CodigoSJ1{2}"
   Circle "Circle_68" at 505,107 size 29x29
      Appearance <- "Var_CodigoSJ1{3}"
   Button "Button_10" at 360,160 size 28x26; TextOff 'Text'
      on Press: SetBit("Panel2CafeJ1")
      on Release: SetBit("Bounce1"); ResetBit("Panel2CafeJ1")
      Appearance <- "Panel2J1Activado"
   Button "Button_11" at 392,160 size 27x26; TextOff 'Text'
      on Press: SetBit("Panel2RosaJ1")
      on Release: SetBit("Bounce1"); ResetBit("Panel2RosaJ1")
      Appearance <- "Panel2J1Activado"
   Button "Button_12" at 424,160 size 27x24; TextOff 'Text'
      on Press: SetBit("Panel2MoradoJ1")
      on Release: SetBit("Bounce1"); ResetBit("Panel2MoradoJ1")
      Appearance <- "Panel2J1Activado"
   Button "Button_13" at 458,160 size 25x25; TextOff 'Text'
      on Press: SetBit("Panel2RojoJ1")
      on Release: SetBit("Bounce1"); ResetBit("Panel2RojoJ1")
      Appearance <- "Panel2J1Activado"
   Button "Button_14" at 489,160 size 25x24; TextOff 'Text'
      on Press: SetBit("Panel2AzulJ1")
      on Release: SetBit("Bounce1"); ResetBit("Panel2AzulJ1")
      Appearance <- "Panel2J1Activado"
   Button "Button_16" at 520,160 size 25x25; TextOff 'Text'
      on Press: SetBit("Panel2VerdeJ1")
      on Release: SetBit("Bounce1"); ResetBit("Panel2VerdeJ1")
      Appearance <- "Panel2J1Activado"
   Button "Button_17" at 549,161 size 25x23; TextOff 'Text'
      on Press: SetBit("Panel2AmarilloJ1")
      on Release: SetBit("Bounce1"); ResetBit("Panel2AmarilloJ1")
      Appearance <- "Panel2J1Activado"
   Circle "Circle_69" at 342,274 size 29x29
      Appearance <- "Var_CodigoOJ1{0}"
   Circle "Circle_70" at 379,274 size 29x29
      Appearance <- "Var_CodigoOJ1{1}"
   Circle "Circle_71" at 416,274 size 29x29
      Appearance <- "Var_CodigoOJ1{2}"
   Circle "Circle_72" at 453,274 size 29x29
      Appearance <- "Var_CodigoOJ1{3}"
   TextField "Text field_11" at 341,233 size 142x23; Text 'Codigo Secreto'
   Button "Button_18" at 621,289 size 135x35; TextOff 'Reiniciar Juego'
      on Press: SetBit("ReiniciarJuego")
      on Release: ResetBit("ReiniciarJuego")
   Rectangle "Rectangle_23" at 401,90 size 13x8
      Appearance <- "Var_CodigoSJ1{0}"
   Rectangle "Rectangle_24" at 438,90 size 13x8
      Appearance <- "Var_CodigoSJ1{1}"
   Rectangle "Rectangle_25" at 475,90 size 13x8
      Appearance <- "Var_CodigoSJ1{2}"
   Rectangle "Rectangle_26" at 512,90 size 13x8
      Appearance <- "Var_CodigoSJ1{3}"
   TextField "Text field_12" at 626,28 size 120x17; Text '1. Selecciona un codigo'
      Visibility <- "Var_VectorMensajes{0}"
   TextField "Text field_13" at 627,48 size 117x43; Text '2. Esperando a que el otro jugador seleccione tu codigo'
      Visibility <- "Var_VectorMensajes{1}"
   TextField "Text field_14" at 625,94 size 130x30; Text '3. Ambos codigos seleccionados. Preparate!'
      Visibility <- "Var_VectorMensajes{2}"
   TextField "Text field_15" at 678,126 size 14x20; Text '5'
      Visibility <- "Var_VectorMensajes{3}"
   TextField "Text field_16" at 678,143 size 14x20; Text '4'
      Visibility <- "Var_VectorMensajes{4}"
   TextField "Text field_17" at 679,160 size 14x20; Text '3'
      Visibility <- "Var_VectorMensajes{5}"
   TextField "Text field_18" at 679,178 size 14x20; Text '2'
      Visibility <- "Var_VectorMensajes{6}"
   TextField "Text field_19" at 679,195 size 14x20; Text '1'
      Visibility <- "Var_VectorMensajes{7}"
   TextField "Text field_20" at 632,219 size 119x43; Text '4. Encuentra el codigo secreto antes que tu oponente!'
      Visibility <- "Var_VectorMensajes{8}"
   TextField "Text field_21" at 501,241 size 101x22; Text 'GANASTE!!!'
      Visibility <- "Var_VectorMensajes{9}"
   TextField "Text field_22" at 503,280 size 108x22; Text 'PERDISTE :('
      Visibility <- "Var_VectorMensajes{10}"
   Rectangle "Rectangle_28" at 322,262 size 178x58
      Visibility <- "DescubrirCodigoSecreto"

Template "Template_1" 800x442
   Button "Exit" at 720,360 size 78x58; TextOff 'Exit'; PictureOff "ExitRuntime_TP700_Comfort_TR"; PictureOn "ExitRuntime_TP700_Comfort_TR"
      on Release: StopRuntime(0)
   Button "Template_Button" at 640,360 size 78x58; TextOff 'Text'
   Button "Template_Button_1" at 560,360 size 78x58; TextOff 'Text'
   Button "Template_Button_2" at 480,360 size 78x58; TextOff 'Text'
   Button "Template_Button_3" at 400,360 size 78x58; TextOff 'Text'
   Button "Template_Button_4" at 321,360 size 78x58; TextOff 'Text'
   Button "Template_Button_5" at 241,360 size 78x58; TextOff 'Text'
   Button "Template_Button_6" at 161,360 size 78x58; TextOff 'Text'
   Button "Alarms" at 81,360 size 78x58; TextOff 'Alarms'; PictureOff "AlarmDisplay_TP700_Comfort_TR"; PictureOn "AlarmDisplay_TP700_Comfort_TR"
      on Release: function_ef3f5d25("Alarm window_Unacknowledged", -1)
   Button "Start screen" at 1,360 size 78x58; TextOff 'Start screen'; PictureOff "NavigateHome_TP700_Comfort_TR"; PictureOn "NavigateHome_TP700_Comfort_TR"
      on Release: ActivateScreen("Root screen", 0)
*)

(* ===== HMI "HMI_RT_2" =====
system functions are stored by id; their names below are inferred from use
connection "HMI_Connection_2": ETHERNET, S7_1500_OMS

HMI tags "Default tag table"
   "Tag_ScreenNumber" : UInt, internal
   "ReiniciarJuego" : Bool = PLC ReiniciarJuego AT %M6.0, 1 s
   "Panel2CafeJ1" : Bool = PLC Panel2CafeJ1 AT %M10.4, 1 s
   "Panel2RosaJ1" : Bool = PLC Panel2RosaJ1 AT %M10.5, 1 s
   "Panel2MoradoJ1" : Bool = PLC Panel2MoradoJ1 AT %M10.6, 1 s
   "Panel2RojoJ1" : Bool = PLC Panel2RojoJ1 AT %M10.7, 1 s
   "Panel2AzulJ1" : Bool = PLC Panel2AzulJ1 AT %M11.0, 1 s
   "Panel2VerdeJ1" : Bool = PLC Panel2VerdeJ1 AT %M11.1, 1 s
   "Panel2AmarilloJ1" : Bool = PLC Panel2AmarilloJ1 AT %M11.2, 1 s
   "Panel1CafeJ1" : Bool = PLC Panel1CafeJ1 AT %M9.5, 1 s
   "Panel1RosaJ1" : Bool = PLC Panel1RosaJ1 AT %M9.6, 1 s
   "Panel1MoradoJ1" : Bool = PLC Panel1MoradoJ1 AT %M9.7, 1 s
   "Panel1RojoJ1" : Bool = PLC Panel1RojoJ1 AT %M10.0, 1 s
   "Panel1AzulJ1" : Bool = PLC Panel1AzulJ1 AT %M10.1, 1 s
   "Panel1VerdeJ1" : Bool = PLC Panel1VerdeJ1 AT %M10.2, 1 s
   "Panel1AmarilloJ1" : Bool = PLC Panel1AmarilloJ1 AT %M10.3, 1 s
   "Panel1J1Activado" : Bool = PLC Panel1J1Activado AT %M13.1, 1 s
   "Panel2J1Activado" : Bool = PLC Panel2J1Activado AT %M13.2, 1 s
   "Var_VectorMensajes{0}" : Int = PLC "Var".VectorMensajes[0], 1 s
   "Var_VectorMensajes{1}" : Int = PLC "Var".VectorMensajes[1], 1 s
   "Var_VectorMensajes{2}" : Int = PLC "Var".VectorMensajes[2], 1 s
   "Var_VectorMensajes{3}" : Int = PLC "Var".VectorMensajes[3], 1 s
   "Var_VectorMensajes{4}" : Int = PLC "Var".VectorMensajes[4], 1 s
   "Var_VectorMensajes{5}" : Int = PLC "Var".VectorMensajes[5], 1 s
   "Var_VectorMensajes{6}" : Int = PLC "Var".VectorMensajes[6], 1 s
   "Var_VectorMensajes{7}" : Int = PLC "Var".VectorMensajes[7], 1 s
   "Var_VectorMensajes{8}" : Int = PLC "Var".VectorMensajes[8], 1 s
   "Var_VectorMensajes{9}" : Int = PLC "Var".VectorMensajes[9], 1 s
   "Var_VectorMensajes{10}" : Int = PLC "Var".VectorMensajes[10], 1 s
   "Var_CodigoOJ1{0}" : Int = PLC "Var".CodigoOJ1[0], 1 s
   "Var_CodigoOJ1{1}" : Int = PLC "Var".CodigoOJ1[1], 1 s
   "Var_CodigoOJ1{2}" : Int = PLC "Var".CodigoOJ1[2], 1 s
   "Var_CodigoOJ1{3}" : Int = PLC "Var".CodigoOJ1[3], 1 s
   "Var_CodigoSJ1{0}" : Int = PLC "Var".CodigoSJ1[0], 1 s
   "Var_CodigoSJ1{1}" : Int = PLC "Var".CodigoSJ1[1], 1 s
   "Var_CodigoSJ1{2}" : Int = PLC "Var".CodigoSJ1[2], 1 s
   "Var_CodigoSJ1{3}" : Int = PLC "Var".CodigoSJ1[3], 1 s
   "Var_VectorPrincipalJ1{0,0}" : Int = PLC "Var".VectorPrincipalJ1[0,0], 1 s
   "Var_VectorPrincipalJ1{0,1}" : Int = PLC "Var".VectorPrincipalJ1[0,1], 1 s
   "Var_VectorPrincipalJ1{0,2}" : Int = PLC "Var".VectorPrincipalJ1[0,2], 1 s
   "Var_VectorPrincipalJ1{0,3}" : Int = PLC "Var".VectorPrincipalJ1[0,3], 1 s
   "Var_VectorPrincipalJ1{1,0}" : Int = PLC "Var".VectorPrincipalJ1[1,0], 1 s
   "Var_VectorPrincipalJ1{1,1}" : Int = PLC "Var".VectorPrincipalJ1[1,1], 1 s
   "Var_VectorPrincipalJ1{1,2}" : Int = PLC "Var".VectorPrincipalJ1[1,2], 1 s
   "Var_VectorPrincipalJ1{1,3}" : Int = PLC "Var".VectorPrincipalJ1[1,3], 1 s
   "Var_VectorPrincipalJ1{2,0}" : Int = PLC "Var".VectorPrincipalJ1[2,0], 1 s
   "Var_VectorPrincipalJ1{2,1}" : Int = PLC "Var".VectorPrincipalJ1[2,1], 1 s
   "Var_VectorPrincipalJ1{2,2}" : Int = PLC "Var".VectorPrincipalJ1[2,2], 1 s
   "Var_VectorPrincipalJ1{2,3}" : Int = PLC "Var".VectorPrincipalJ1[2,3], 1 s
   "Var_VectorPrincipalJ1{3,0}" : Int = PLC "Var".VectorPrincipalJ1[3,0], 1 s
   "Var_VectorPrincipalJ1{3,1}" : Int = PLC "Var".VectorPrincipalJ1[3,1], 1 s
   "Var_VectorPrincipalJ1{3,2}" : Int = PLC "Var".VectorPrincipalJ1[3,2], 1 s
   "Var_VectorPrincipalJ1{3,3}" : Int = PLC "Var".VectorPrincipalJ1[3,3], 1 s
   "Var_VectorPrincipalJ1{4,0}" : Int = PLC "Var".VectorPrincipalJ1[4,0], 1 s
   "Var_VectorPrincipalJ1{4,1}" : Int = PLC "Var".VectorPrincipalJ1[4,1], 1 s
   "Var_VectorPrincipalJ1{4,2}" : Int = PLC "Var".VectorPrincipalJ1[4,2], 1 s
   "Var_VectorPrincipalJ1{4,3}" : Int = PLC "Var".VectorPrincipalJ1[4,3], 1 s
   "Var_VectorPrincipalJ1{5,0}" : Int = PLC "Var".VectorPrincipalJ1[5,0], 1 s
   "Var_VectorPrincipalJ1{5,1}" : Int = PLC "Var".VectorPrincipalJ1[5,1], 1 s
   "Var_VectorPrincipalJ1{5,2}" : Int = PLC "Var".VectorPrincipalJ1[5,2], 1 s
   "Var_VectorPrincipalJ1{5,3}" : Int = PLC "Var".VectorPrincipalJ1[5,3], 1 s
   "Var_VectorPrincipalJ1{6,0}" : Int = PLC "Var".VectorPrincipalJ1[6,0], 1 s
   "Var_VectorPrincipalJ1{6,1}" : Int = PLC "Var".VectorPrincipalJ1[6,1], 1 s
   "Var_VectorPrincipalJ1{6,2}" : Int = PLC "Var".VectorPrincipalJ1[6,2], 1 s
   "Var_VectorPrincipalJ1{6,3}" : Int = PLC "Var".VectorPrincipalJ1[6,3], 1 s
   "Var_VectorPrincipalJ1{7,0}" : Int = PLC "Var".VectorPrincipalJ1[7,0], 1 s
   "Var_VectorPrincipalJ1{7,1}" : Int = PLC "Var".VectorPrincipalJ1[7,1], 1 s
   "Var_VectorPrincipalJ1{7,2}" : Int = PLC "Var".VectorPrincipalJ1[7,2], 1 s
   "Var_VectorPrincipalJ1{7,3}" : Int = PLC "Var".VectorPrincipalJ1[7,3], 1 s
   "Var_VectorSecundarioJ1{0,0}" : Int = PLC "Var".VectorSecundarioJ1[0,0], 1 s
   "Var_VectorSecundarioJ1{0,1}" : Int = PLC "Var".VectorSecundarioJ1[0,1], 1 s
   "Var_VectorSecundarioJ1{0,2}" : Int = PLC "Var".VectorSecundarioJ1[0,2], 1 s
   "Var_VectorSecundarioJ1{0,3}" : Int = PLC "Var".VectorSecundarioJ1[0,3], 1 s
   "Var_VectorSecundarioJ1{1,0}" : Int = PLC "Var".VectorSecundarioJ1[1,0], 1 s
   "Var_VectorSecundarioJ1{1,1}" : Int = PLC "Var".VectorSecundarioJ1[1,1], 1 s
   "Var_VectorSecundarioJ1{1,2}" : Int = PLC "Var".VectorSecundarioJ1[1,2], 1 s
   "Var_VectorSecundarioJ1{1,3}" : Int = PLC "Var".VectorSecundarioJ1[1,3], 1 s
   "Var_VectorSecundarioJ1{2,0}" : Int = PLC "Var".VectorSecundarioJ1[2,0], 1 s
   "Var_VectorSecundarioJ1{2,1}" : Int = PLC "Var".VectorSecundarioJ1[2,1], 1 s
   "Var_VectorSecundarioJ1{2,2}" : Int = PLC "Var".VectorSecundarioJ1[2,2], 1 s
   "Var_VectorSecundarioJ1{2,3}" : Int = PLC "Var".VectorSecundarioJ1[2,3], 1 s
   "Var_VectorSecundarioJ1{3,0}" : Int = PLC "Var".VectorSecundarioJ1[3,0], 1 s
   "Var_VectorSecundarioJ1{3,1}" : Int = PLC "Var".VectorSecundarioJ1[3,1], 1 s
   "Var_VectorSecundarioJ1{3,2}" : Int = PLC "Var".VectorSecundarioJ1[3,2], 1 s
   "Var_VectorSecundarioJ1{3,3}" : Int = PLC "Var".VectorSecundarioJ1[3,3], 1 s
   "Var_VectorSecundarioJ1{4,0}" : Int = PLC "Var".VectorSecundarioJ1[4,0], 1 s
   "Var_VectorSecundarioJ1{4,1}" : Int = PLC "Var".VectorSecundarioJ1[4,1], 1 s
   "Var_VectorSecundarioJ1{4,2}" : Int = PLC "Var".VectorSecundarioJ1[4,2], 1 s
   "Var_VectorSecundarioJ1{4,3}" : Int = PLC "Var".VectorSecundarioJ1[4,3], 1 s
   "Var_VectorSecundarioJ1{5,0}" : Int = PLC "Var".VectorSecundarioJ1[5,0], 1 s
   "Var_VectorSecundarioJ1{5,1}" : Int = PLC "Var".VectorSecundarioJ1[5,1], 1 s
   "Var_VectorSecundarioJ1{5,2}" : Int = PLC "Var".VectorSecundarioJ1[5,2], 1 s
   "Var_VectorSecundarioJ1{5,3}" : Int = PLC "Var".VectorSecundarioJ1[5,3], 1 s
   "Var_VectorSecundarioJ1{6,0}" : Int = PLC "Var".VectorSecundarioJ1[6,0], 1 s
   "Var_VectorSecundarioJ1{6,1}" : Int = PLC "Var".VectorSecundarioJ1[6,1], 1 s
   "Var_VectorSecundarioJ1{6,2}" : Int = PLC "Var".VectorSecundarioJ1[6,2], 1 s
   "Var_VectorSecundarioJ1{6,3}" : Int = PLC "Var".VectorSecundarioJ1[6,3], 1 s
   "Var_VectorSecundarioJ1{7,0}" : Int = PLC "Var".VectorSecundarioJ1[7,0], 1 s
   "Var_VectorSecundarioJ1{7,1}" : Int = PLC "Var".VectorSecundarioJ1[7,1], 1 s
   "Var_VectorSecundarioJ1{7,2}" : Int = PLC "Var".VectorSecundarioJ1[7,2], 1 s
   "Var_VectorSecundarioJ1{7,3}" : Int = PLC "Var".VectorSecundarioJ1[7,3], 1 s
   "Bounce1" : Bool = PLC Bounce1 AT %M13.6, 1 s
   "Bounce5" : Bool = PLC Bounce5 AT %M14.1, 1 s
   "ReiniciarCorrSimiDisp" : Bool = PLC ReiniciarCorrSimiDisp AT %M34.0, 1 s
   "Panel2J2Activado" : Bool = PLC Panel2J2Activado AT %M13.4, 1 s
   "Var_CodigoSJ2{0}" : Int = PLC "Var".CodigoSJ2[0], 1 s
   "Var_CodigoSJ2{1}" : Int = PLC "Var".CodigoSJ2[1], 1 s
   "Var_CodigoSJ2{2}" : Int = PLC "Var".CodigoSJ2[2], 1 s
   "Var_CodigoSJ2{3}" : Int = PLC "Var".CodigoSJ2[3], 1 s
   "Panel2CafeJ2" : Bool = PLC Panel2CafeJ2 AT %M12.2, 1 s
   "Var_CodigoOJ2{0}" : Int = PLC "Var".CodigoOJ2[0], 1 s
   "Var_CodigoOJ2{1}" : Int = PLC "Var".CodigoOJ2[1], 1 s
   "Var_CodigoOJ2{2}" : Int = PLC "Var".CodigoOJ2[2], 1 s
   "Var_CodigoOJ2{3}" : Int = PLC "Var".CodigoOJ2[3], 1 s
   "Bounce6" : Bool = PLC Bounce6 AT %M14.2, 1 s
   "Panel2RosaJ2" : Bool = PLC Panel2RosaJ2 AT %M12.3, 1 s
   "Panel2MoradoJ2" : Bool = PLC Panel2MoradoJ2 AT %M12.4, 1 s
   "Panel2RojoJ2" : Bool = PLC Panel2RojoJ2 AT %M12.5, 1 s
   "Panel2AzulJ2" : Bool = PLC Panel2AzulJ2 AT %M12.6, 1 s
   "Panel2VerdeJ2" : Bool = PLC Panel2VerdeJ2 AT %M12.7, 1 s
   "Panel2AmarilloJ2" : Bool = PLC Panel2AmarilloJ2 AT %M13.0, 1 s
   "Var_VectorMensajesJ2{0}" : Int = PLC "Var".VectorMensajesJ2[0], 1 s
   "Var_VectorMensajesJ2{1}" : Int = PLC "Var".VectorMensajesJ2[1], 1 s
   "Var_VectorMensajesJ2{2}" : Int = PLC "Var".VectorMensajesJ2[2], 1 s
   "Var_VectorMensajesJ2{3}" : Int = PLC "Var".VectorMensajesJ2[3], 1 s
   "Var_VectorMensajesJ2{4}" : Int = PLC "Var".VectorMensajesJ2[4], 1 s
   "Var_VectorMensajesJ2{5}" : Int = PLC "Var".VectorMensajesJ2[5], 1 s
   "Var_VectorMensajesJ2{6}" : Int = PLC "Var".VectorMensajesJ2[6], 1 s
   "Var_VectorMensajesJ2{7}" : Int = PLC "Var".VectorMensajesJ2[7], 1 s
   "Var_VectorMensajesJ2{8}" : Int = PLC "Var".VectorMensajesJ2[8], 1 s
   "Var_VectorMensajesJ2{9}" : Int = PLC "Var".VectorMensajesJ2[9], 1 s
   "Var_VectorMensajesJ2{10}" : Int = PLC "Var".VectorMensajesJ2[10], 1 s
   "Panel1J2Activado" : Bool = PLC Panel1J2Activado AT %M13.3, 1 s
   "Panel1CafeJ2" : Bool = PLC Panel1CafeJ2 AT %M11.3, 1 s
   "Bounce10" : Bool = PLC Bounce10 AT %M14.5, 1 s
   "Panel1RosaJ2" : Bool = PLC Panel1RosaJ2 AT %M11.4, 1 s
   "Panel1MoradoJ2" : Bool = PLC Panel1MoradoJ2 AT %M11.5, 1 s
   "Panel1AzulJ2" : Bool = PLC Panel1AzulJ2 AT %M11.7, 1 s
   "Panel1VerdeJ2" : Bool = PLC Panel1VerdeJ2 AT %M12.0, 1 s
   "Panel1AmarilloJ2" : Bool = PLC Panel1AmarilloJ2 AT %M12.1, 1 s
   "Var_VectorPrincipalJ2{0,0}" : Int = PLC "Var".VectorPrincipalJ2[0,0], 1 s
   "Var_VectorPrincipalJ2{0,1}" : Int = PLC "Var".VectorPrincipalJ2[0,1], 1 s
   "Var_VectorPrincipalJ2{0,2}" : Int = PLC "Var".VectorPrincipalJ2[0,2], 1 s
   "Var_VectorPrincipalJ2{0,3}" : Int = PLC "Var".VectorPrincipalJ2[0,3], 1 s
   "Var_VectorPrincipalJ2{1,0}" : Int = PLC "Var".VectorPrincipalJ2[1,0], 1 s
   "Var_VectorPrincipalJ2{1,1}" : Int = PLC "Var".VectorPrincipalJ2[1,1], 1 s
   "Var_VectorPrincipalJ2{1,2}" : Int = PLC "Var".VectorPrincipalJ2[1,2], 1 s
   "Var_VectorPrincipalJ2{1,3}" : Int = PLC "Var".VectorPrincipalJ2[1,3], 1 s
   "Var_VectorPrincipalJ2{2,0}" : Int = PLC "Var".VectorPrincipalJ2[2,0], 1 s
   "Var_VectorPrincipalJ2{2,1}" : Int = PLC "Var".VectorPrincipalJ2[2,1], 1 s
   "Var_VectorPrincipalJ2{2,2}" : Int = PLC "Var".VectorPrincipalJ2[2,2], 1 s
   "Var_VectorPrincipalJ2{2,3}" : Int = PLC "Var".VectorPrincipalJ2[2,3], 1 s
   "Var_VectorPrincipalJ2{3,0}" : Int = PLC "Var".VectorPrincipalJ2[3,0], 1 s
   "Var_VectorPrincipalJ2{3,1}" : Int = PLC "Var".VectorPrincipalJ2[3,1], 1 s
   "Var_VectorPrincipalJ2{3,2}" : Int = PLC "Var".VectorPrincipalJ2[3,2], 1 s
   "Var_VectorPrincipalJ2{3,3}" : Int = PLC "Var".VectorPrincipalJ2[3,3], 1 s
   "Var_VectorPrincipalJ2{4,0}" : Int = PLC "Var".VectorPrincipalJ2[4,0], 1 s
   "Var_VectorPrincipalJ2{4,1}" : Int = PLC "Var".VectorPrincipalJ2[4,1], 1 s
   "Var_VectorPrincipalJ2{4,2}" : Int = PLC "Var".VectorPrincipalJ2[4,2], 1 s
   "Var_VectorPrincipalJ2{4,3}" : Int = PLC "Var".VectorPrincipalJ2[4,3], 1 s
   "Var_VectorPrincipalJ2{5,0}" : Int = PLC "Var".VectorPrincipalJ2[5,0], 1 s
   "Var_VectorPrincipalJ2{5,1}" : Int = PLC "Var".VectorPrincipalJ2[5,1], 1 s
   "Var_VectorPrincipalJ2{5,2}" : Int = PLC "Var".VectorPrincipalJ2[5,2], 1 s
   "Var_VectorPrincipalJ2{5,3}" : Int = PLC "Var".VectorPrincipalJ2[5,3], 1 s
   "Var_VectorPrincipalJ2{6,0}" : Int = PLC "Var".VectorPrincipalJ2[6,0], 1 s
   "Var_VectorPrincipalJ2{6,1}" : Int = PLC "Var".VectorPrincipalJ2[6,1], 1 s
   "Var_VectorPrincipalJ2{6,2}" : Int = PLC "Var".VectorPrincipalJ2[6,2], 1 s
   "Var_VectorPrincipalJ2{6,3}" : Int = PLC "Var".VectorPrincipalJ2[6,3], 1 s
   "Var_VectorPrincipalJ2{7,0}" : Int = PLC "Var".VectorPrincipalJ2[7,0], 1 s
   "Var_VectorPrincipalJ2{7,1}" : Int = PLC "Var".VectorPrincipalJ2[7,1], 1 s
   "Var_VectorPrincipalJ2{7,2}" : Int = PLC "Var".VectorPrincipalJ2[7,2], 1 s
   "Var_VectorPrincipalJ2{7,3}" : Int = PLC "Var".VectorPrincipalJ2[7,3], 1 s
   "Var_VectorSecundarioJ2{0,2}" : Int = PLC "Var".VectorSecundarioJ2[0,2], 1 s
   "Var_VectorSecundarioJ2{0,3}" : Int = PLC "Var".VectorSecundarioJ2[0,3], 1 s
   "Var_VectorSecundarioJ2{0,0}" : Int = PLC "Var".VectorSecundarioJ2[0,0], 1 s
   "Var_VectorSecundarioJ2{0,1}" : Int = PLC "Var".VectorSecundarioJ2[0,1], 1 s
   "Var_VectorSecundarioJ2{1,0}" : Int = PLC "Var".VectorSecundarioJ2[1,0], 1 s
   "Var_VectorSecundarioJ2{1,1}" : Int = PLC "Var".VectorSecundarioJ2[1,1], 1 s
   "Var_VectorSecundarioJ2{1,2}" : Int = PLC "Var".VectorSecundarioJ2[1,2], 1 s
   "Var_VectorSecundarioJ2{1,3}" : Int = PLC "Var".VectorSecundarioJ2[1,3], 1 s
   "Var_VectorSecundarioJ2{2,0}" : Int = PLC "Var".VectorSecundarioJ2[2,0], 1 s
   "Var_VectorSecundarioJ2{2,1}" : Int = PLC "Var".VectorSecundarioJ2[2,1], 1 s
   "Var_VectorSecundarioJ2{2,2}" : Int = PLC "Var".VectorSecundarioJ2[2,2], 1 s
   "Var_VectorSecundarioJ2{2,3}" : Int = PLC "Var".VectorSecundarioJ2[2,3], 1 s
   "Var_VectorSecundarioJ2{3,0}" : Int = PLC "Var".VectorSecundarioJ2[3,0], 1 s
   "Var_VectorSecundarioJ2{3,1}" : Int = PLC "Var".VectorSecundarioJ2[3,1], 1 s
   "Var_VectorSecundarioJ2{3,2}" : Int = PLC "Var".VectorSecundarioJ2[3,2], 1 s
   "Var_VectorSecundarioJ2{3,3}" : Int = PLC "Var".VectorSecundarioJ2[3,3], 1 s
   "Var_VectorSecundarioJ2{4,0}" : Int = PLC "Var".VectorSecundarioJ2[4,0], 1 s
   "Var_VectorSecundarioJ2{4,1}" : Int = PLC "Var".VectorSecundarioJ2[4,1], 1 s
   "Var_VectorSecundarioJ2{4,2}" : Int = PLC "Var".VectorSecundarioJ2[4,2], 1 s
   "Var_VectorSecundarioJ2{4,3}" : Int = PLC "Var".VectorSecundarioJ2[4,3], 1 s
   "Var_VectorSecundarioJ2{5,0}" : Int = PLC "Var".VectorSecundarioJ2[5,0], 1 s
   "Var_VectorSecundarioJ2{5,1}" : Int = PLC "Var".VectorSecundarioJ2[5,1], 1 s
   "Var_VectorSecundarioJ2{5,2}" : Int = PLC "Var".VectorSecundarioJ2[5,2], 1 s
   "Var_VectorSecundarioJ2{5,3}" : Int = PLC "Var".VectorSecundarioJ2[5,3], 1 s
   "Var_VectorSecundarioJ2{6,0}" : Int = PLC "Var".VectorSecundarioJ2[6,0], 1 s
   "Var_VectorSecundarioJ2{6,1}" : Int = PLC "Var".VectorSecundarioJ2[6,1], 1 s
   "Var_VectorSecundarioJ2{6,2}" : Int = PLC "Var".VectorSecundarioJ2[6,2], 1 s
   "Var_VectorSecundarioJ2{6,3}" : Int = PLC "Var".VectorSecundarioJ2[6,3], 1 s
   "Var_VectorSecundarioJ2{7,0}" : Int = PLC "Var".VectorSecundarioJ2[7,0], 1 s
   "Var_VectorSecundarioJ2{7,1}" : Int = PLC "Var".VectorSecundarioJ2[7,1], 1 s
   "Var_VectorSecundarioJ2{7,2}" : Int = PLC "Var".VectorSecundarioJ2[7,2], 1 s
   "Var_VectorSecundarioJ2{7,3}" : Int = PLC "Var".VectorSecundarioJ2[7,3], 1 s
   "DescubrirCodigoSecreto" : Bool = PLC DescubrirCodigoSecreto AT %M50.3, 1 s
   "Panel1RojoJ2" : Bool = PLC Panel1RojoJ2 AT %M11.6, 1 s

screen "Root screen" 800x442, template "Template_1"
   on GenerateScreen: SetTag("Tag_ScreenNumber", 1)
   Button "Button_3" at 67,293 size 28x26; TextOff 'Text'
      on Release: SetBit("Bounce10"); ResetBit("Panel1CafeJ2")
      on Press: SetBit("Panel1CafeJ2")
      Appearance <- "Panel1J2Activado"
   Button "Button_4" at 99,293 size 27x26; TextOff 'Text'
      on Release: SetBit("Bounce10"); ResetBit("Panel1RosaJ2")
      on Press: SetBit("Panel1RosaJ2")
      Appearance <- "Panel1J2Activado"
   Button "Button_5" at 131,293 size 27x24; TextOff 'Text'
      on Release: SetBit("Bounce10"); ResetBit("Panel1MoradoJ2")
      on Press: SetBit("Panel1MoradoJ2")
      Appearance <- "Panel1J2Activado"
   Button "Button_6" at 165,293 size 25x25; TextOff 'Text'
      on Release: SetBit("Bounce10"); ResetBit("Panel1RojoJ2")
      on Press: SetBit("Panel1RojoJ2")
      Appearance <- "Panel1J2Activado"
   Button "Button_7" at 196,293 size 25x24; TextOff 'Text'
      on Release: SetBit("Bounce10"); ResetBit("Panel1AzulJ2")
      on Press: SetBit("Panel1AzulJ2")
      Appearance <- "Panel1J2Activado"
   Button "Button_8" at 227,293 size 25x25; TextOff 'Text'
      on Release: SetBit("Bounce10"); ResetBit("Panel1VerdeJ2")
      on Press: SetBit("Panel1VerdeJ2")
      Appearance <- "Panel1J2Activado"
   Button "Button_9" at 256,294 size 25x23; TextOff 'Text'
      on Release: SetBit("Bounce10"); ResetBit("Panel1AmarilloJ2")
      on Press: SetBit("Panel1AmarilloJ2")
      Appearance <- "Panel1J2Activado"
   TextField "Text field_1" at 37,250 size 16x23; Text '1'
   TextField "Text field_2" at 37,221 size 16x23; Text '2'
   TextField "Text field_3" at 37,194 size 16x23; Text '3'
   TextField "Text field_4" at 37,163 size 16x23; Text '4'
   TextField "Text field_5" at 37,134 size 16x23; Text '5'
   TextField "Text field_6" at 37,103 size 16x23; Text '6'
   TextField "Text field_7" at 37,74 size 16x23; Text '7'
   TextField "Text field_8" at 37,43 size 16x23; Text '8'
   Circle "Circle_1" at 92,254 size 23x23
      Appearance <- "Var_VectorPrincipalJ2{0,0}"
   Circle "Circle_2" at 128,254 size 23x23
      Appearance <- "Var_VectorPrincipalJ2{0,1}"
   Circle "Circle_3" at 164,254 size 23x23
      Appearance <- "Var_VectorPrincipalJ2{0,2}"
   Circle "Circle_4" at 201,254 size 23x23
      Appearance <- "Var_VectorPrincipalJ2{0,3}"
   Circle "Circle_5" at 92,224 size 23x23
      Appearance <- "Var_VectorPrincipalJ2{1,0}"
   Circle "Circle_6" at 128,224 size 23x23
      Appearance <- "Var_VectorPrincipalJ2{1,1}"
   Circle "Circle_7" at 164,224 size 23x23
      Appearance <- "Var_VectorPrincipalJ2{1,2}"
   Circle "Circle_8" at 201,224 size 23x23
      Appearance <- "Var_VectorPrincipalJ2{1,3}"
   Circle "Circle_9" at 92,194 size 23x23
      Appearance <- "Var_VectorPrincipalJ2{2,0}"
   Circle "Circle_10" at 128,194 size 23x23
      Appearance <- "Var_VectorPrincipalJ2{2,1}"
   Circle "Circle_11" at 164,194 size 23x23
      Appearance <- "Var_VectorPrincipalJ2{2,2}"
   Circle "Circle_12" at 201,194 size 23x23
      Appearance <- "Var_VectorPrincipalJ2{2,3}"
   Circle "Circle_13" at 92,164 size 23x23
      Appearance <- "Var_VectorPrincipalJ2{3,0}"
   Circle "Circle_14" at 128,164 size 23x23
      Appearance <- "Var_VectorPrincipalJ2{3,1}"
   Circle "Circle_15" at 164,164 size 23x23
      Appearance <- "Var_VectorPrincipalJ2{3,2}"
   Circle "Circle_16" at 201,164 size 23x23
      Appearance <- "Var_VectorPrincipalJ2{3,3}"
   Circle "Circle_17" at 92,134 size 23x23
      Appearance <- "Var_VectorPrincipalJ2{4,0}"
   Circle "Circle_18" at 128,134 size 23x23
      Appearance <- "Var_VectorPrincipalJ2{4,1}"
   Circle "Circle_19" at 164,134 size 23x23
      Appearance <- "Var_VectorPrincipalJ2{4,2}"
   Circle "Circle_20" at 201,134 size 23x23
      Appearance <- "Var_VectorPrincipalJ2{4,3}"
   Circle "Circle_21" at 92,104 size 23x23
      Appearance <- "Var_VectorPrincipalJ2{5,0}"
   Circle "Circle_22" at 128,104 size 23x23
      Appearance <- "Var_VectorPrincipalJ2{5,1}"
   Circle "Circle_23" at 164,104 size 23x23
      Appearance <- "Var_VectorPrincipalJ2{5,2}"
   Circle "Circle_24" at 201,104 size 23x23
      Appearance <- "Var_VectorPrincipalJ2{5,3}"
   Circle "Circle_25" at 92,74 size 23x23
      Appearance <- "Var_VectorPrincipalJ2{6,0}"
   Circle "Circle_26" at 128,74 size 23x23
      Appearance <- "Var_VectorPrincipalJ2{6,1}"
   Circle "Circle_27" at 164,74 size 23x23
      Appearance <- "Var_VectorPrincipalJ2{6,2}"
   Circle "Circle_28" at 201,74 size 23x23
      Appearance <- "Var_VectorPrincipalJ2{6,3}"
   Circle "Circle_29" at 92,44 size 23x23
      Appearance <- "Var_VectorPrincipalJ2{7,0}"
   Circle "Circle_30" at 128,44 size 23x23
      Appearance <- "Var_VectorPrincipalJ2{7,1}"
   Circle "Circle_31" at 164,44 size 23x23
      Appearance <- "Var_VectorPrincipalJ2{7,2}"
   Circle "Circle_32" at 201,44 size 23x23
      Appearance <- "Var_VectorPrincipalJ2{7,3}"
   Circle "Circle_33" at 255,253 size 14x14
      Appearance <- "Var_VectorSecundarioJ2{0,0}"
   Circle "Circle_34" at 270,253 size 14x14
      Appearance <- "Var_VectorSecundarioJ2{0,1}"
   Circle "Circle_35" at 255,267 size 14x14
      Appearance <- "Var_VectorSecundarioJ2{0,2}"
   Circle "Circle_36" at 270,267 size 14x14
      Appearance <- "Var_VectorSecundarioJ2{0,3}"
   Circle "Circle_37" at 255,223 size 14x14
      Appearance <- "Var_VectorSecundarioJ2{1,0}"
   Circle "Circle_38" at 270,223 size 14x14
      Appearance <- "Var_VectorSecundarioJ2{1,1}"
   Circle "Circle_39" at 255,237 size 14x14
      Appearance <- "Var_VectorSecundarioJ2{1,2}"
   Circle "Circle_40" at 270,237 size 14x14
      Appearance <- "Var_VectorSecundarioJ2{1,3}"
   Circle "Circle_41" at 255,193 size 14x14
      Appearance <- "Var_VectorSecundarioJ2{2,0}"
   Circle "Circle_42" at 270,193 size 14x14
      Appearance <- "Var_VectorSecundarioJ2{2,1}"
   Circle "Circle_43" at 255,207 size 14x14
      Appearance <- "Var_VectorSecundarioJ2{2,2}"
   Circle "Circle_44" at 270,207 size 14x14
      Appearance <- "Var_VectorSecundarioJ2{2,3}"
   Circle "Circle_45" at 255,163 size 14x14
      Appearance <- "Var_VectorSecundarioJ2{3,0}"
   Circle "Circle_46" at 270,163 size 14x14
      Appearance <- "Var_VectorSecundarioJ2{3,1}"
   Circle "Circle_47" at 255,177 size 14x14
      Appearance <- "Var_VectorSecundarioJ2{3,2}"
   Circle "Circle_48" at 270,177 size 14x14
      Appearance <- "Var_VectorSecundarioJ2{3,3}"
   Circle "Circle_49" at 255,133 size 14x14
      Appearance <- "Var_VectorSecundarioJ2{4,0}"
   Circle "Circle_50" at 270,133 size 14x14
      Appearance <- "Var_VectorSecundarioJ2{4,1}"
   Circle "Circle_51" at 255,147 size 14x14
      Appearance <- "Var_VectorSecundarioJ2{4,2}"
   Circle "Circle_52" at 270,147 size 14x14
      Appearance <- "Var_VectorSecundarioJ2{4,3}"
   Circle "Circle_53" at 255,103 size 14x14
      Appearance <- "Var_VectorSecundarioJ2{5,0}"
   Circle "Circle_54" at 270,103 size 14x14
      Appearance <- "Var_VectorSecundarioJ2{5,1}"
   Circle "Circle_55" at 255,117 size 14x14
      Appearance <- "Var_VectorSecundarioJ2{5,2}"
   Circle "Circle_56" at 270,117 size 14x14
      Appearance <- "Var_VectorSecundarioJ2{5,3}"
   Circle "Circle_57" at 255,73 size 14x14
      Appearance <- "Var_VectorSecundarioJ2{6,0}"
   Circle "Circle_58" at 270,73 size 14x14
      Appearance <- "Var_VectorSecundarioJ2{6,1}"
   Circle "Circle_59" at 255,87 size 14x14
      Appearance <- "Var_VectorSecundarioJ2{6,2}"
   Circle "Circle_60" at 270,87 size 14x14
      Appearance <- "Var_VectorSecundarioJ2{6,3}"
   Circle "Circle_61" at 255,43 size 14x14
      Appearance <- "Var_VectorSecundarioJ2{7,0}"
   Circle "Circle_62" at 270,43 size 14x14
      Appearance <- "Var_VectorSecundarioJ2{7,1}"
   Circle "Circle_63" at 255,57 size 14x14
      Appearance <- "Var_VectorSecundarioJ2{7,2}"
   Circle "Circle_64" at 270,57 size 14x14
      Appearance <- "Var_VectorSecundarioJ2{7,3}"
   TextField "Text field_9" at 339,40 size 252x42; Text 'Selecciona el Codigo de tu Oponente:'
   TextField "Text field_10" at 388,20 size 166x23; Text 'INICIO Jugador 2'
   Circle "Circle_65" at 393,108 size 29x29
      Appearance <- "Var_CodigoSJ2{0}"
   Circle "Circle_66" at 431,107 size 29x29
      Appearance <- "Var_CodigoSJ2{1}"
   Circle "Circle_67" at 467,108 size 29x29
      Appearance <- "Var_CodigoSJ2{2}"
   Circle "Circle_68" at 505,107 size 29x29
      Appearance <- "Var_CodigoSJ2{3}"
   Button "Button_10" at 360,160 size 28x26; TextOff 'Text'
      on Release: SetBit("Bounce6"); ResetBit("Panel2CafeJ2")
      on Press: SetBit("Panel2CafeJ2")
      Appearance <- "Panel2J2Activado"
   Button "Button_11" at 392,160 size 27x26; TextOff 'Text'
      on Release: SetBit("Bounce6"); ResetBit("Panel2RosaJ2")
      on Press: SetBit("Panel2RosaJ2")
      Appearance <- "Panel2J2Activado"
   Button "Button_12" at 424,160 size 27x24; TextOff 'Text'
      on Release: SetBit("Bounce6"); ResetBit("Panel2MoradoJ2")
      on Press: SetBit("Panel2MoradoJ2")
      Appearance <- "Panel2J2Activado"
   Button "Button_13" at 458,160 size 25x25; TextOff 'Text'
      on Release: SetBit("Bounce6"); ResetBit("Panel2RojoJ2")
      on Press: SetBit("Panel2RojoJ2")
      Appearance <- "Panel2J2Activado"
   Button "Button_14" at 489,160 size 25x24; TextOff 'Text'
      on Release: SetBit("Bounce6"); ResetBit("Panel2AzulJ2")
      on Press: SetBit("Panel2AzulJ2")
      Appearance <- "Panel2J2Activado"
   Button "Button_16" at 520,160 size 25x25; TextOff 'Text'
      on Release: SetBit("Bounce6"); ResetBit("Panel2VerdeJ2")
      on Press: SetBit("Panel2VerdeJ2")
      Appearance <- "Panel2J2Activado"
   Button "Button_17" at 549,161 size 25x23; TextOff 'Text'
      on Release: SetBit("Bounce6"); ResetBit("Panel2AmarilloJ2")
      on Press: SetBit("Panel2AmarilloJ2")
      Appearance <- "Panel2J2Activado"
   Circle "Circle_69" at 342,274 size 29x29
      Appearance <- "Var_CodigoOJ2{0}"
   Circle "Circle_70" at 379,274 size 29x29
      Appearance <- "Var_CodigoOJ2{1}"
   Circle "Circle_71" at 416,274 size 29x29
      Appearance <- "Var_CodigoOJ2{2}"
   Circle "Circle_72" at 453,274 size 29x29
      Appearance <- "Var_CodigoOJ2{3}"
   TextField "Text field_11" at 341,233 size 142x23; Text 'Codigo Secreto'
   Button "Button_18" at 621,289 size 135x35; TextOff 'Reiniciar Juego'
      on Release: ResetBit("ReiniciarJuego")
      on Press: SetBit("ReiniciarJuego")
   Rectangle "Rectangle_23" at 401,90 size 13x8
      Appearance <- "Var_CodigoSJ2{0}"
   Rectangle "Rectangle_24" at 438,90 size 13x8
      Appearance <- "Var_CodigoSJ2{1}"
   Rectangle "Rectangle_25" at 475,90 size 13x8
      Appearance <- "Var_CodigoSJ2{2}"
   Rectangle "Rectangle_26" at 512,90 size 13x8
      Appearance <- "Var_CodigoSJ2{3}"
   TextField "Text field_12" at 626,28 size 120x17; Text '1. Selecciona un codigo'
      Visibility <- "Var_VectorMensajesJ2{0}"
   TextField "Text field_13" at 627,48 size 117x43; Text '2. Esperando a que el otro jugador seleccione tu codigo'
      Visibility <- "Var_VectorMensajesJ2{1}"
   TextField "Text field_14" at 625,94 size 130x30; Text '3. Ambos codigos seleccionados. Preparate!'
      Visibility <- "Var_VectorMensajesJ2{2}"
   TextField "Text field_15" at 678,126 size 14x20; Text '5'
      Visibility <- "Var_VectorMensajesJ2{3}"
   TextField "Text field_16" at 678,143 size 14x20; Text '4'
      Visibility <- "Var_VectorMensajesJ2{4}"
   TextField "Text field_17" at 679,160 size 14x20; Text '3'
      Visibility <- "Var_VectorMensajesJ2{5}"
   TextField "Text field_18" at 679,178 size 14x20; Text '2'
      Visibility <- "Var_VectorMensajesJ2{6}"
   TextField "Text field_19" at 679,195 size 14x20; Text '1'
      Visibility <- "Var_VectorMensajesJ2{7}"
   TextField "Text field_20" at 632,219 size 119x43; Text '4. Encuentra el codigo secreto antes que tu oponente!'
      Visibility <- "Var_VectorMensajesJ2{8}"
   TextField "Text field_21" at 501,241 size 101x22; Text 'GANASTE!!!'
      Visibility <- "Var_VectorMensajesJ2{9}"
   TextField "Text field_22" at 503,280 size 108x22; Text 'PERDISTE :('
      Visibility <- "Var_VectorMensajesJ2{10}"
   Rectangle "Rectangle_28" at 322,262 size 178x58
      Visibility <- "DescubrirCodigoSecreto"

Template "Template_1" 800x442
   Button "Exit" at 720,360 size 78x58; TextOn 'Exit'; TextOff 'Exit'; PictureOn "ExitRuntime_TP700_Comfort_TR"; PictureOff "ExitRuntime_TP700_Comfort_TR"
      on Release: StopRuntime(0)
   Button "Template_Button" at 640,360 size 78x58; TextOff 'Text'
   Button "Template_Button_1" at 560,360 size 78x58; TextOff 'Text'
   Button "Template_Button_2" at 480,360 size 78x58; TextOff 'Text'
   Button "Template_Button_3" at 400,360 size 78x58; TextOff 'Text'
   Button "Template_Button_4" at 321,360 size 78x58; TextOff 'Text'
   Button "Template_Button_5" at 241,360 size 78x58; TextOff 'Text'
   Button "Template_Button_6" at 161,360 size 78x58; TextOff 'Text'
   Button "Alarms" at 81,360 size 78x58; TextOn 'Alarms'; TextOff 'Alarms'; PictureOn "AlarmDisplay_TP700_Comfort_TR"; PictureOff "AlarmDisplay_TP700_Comfort_TR"
      on Release: function_ef3f5d25("Alarm window_Unacknowledged", -1)
   Button "Start screen" at 1,360 size 78x58; TextOn 'Start screen'; TextOff 'Start screen'; PictureOn "NavigateHome_TP700_Comfort_TR"; PictureOff "NavigateHome_TP700_Comfort_TR"
      on Release: ActivateScreen("Root screen", 0)
*)